(* IEC 61131-3 sources: Industry-PLC-LLM/data/PLCBEAD_repo/PLCBEAD_PLCEmbed-main/PLC-BEAD/Source/OpenPLCv2 (part 5) *)

(* ---- FT_DERIV.ST ---- *)
FUNCTION_BLOCK T_PLC_US_Block
	VAR_OUTPUT
		T_PLC_US :	UDINT;
	END_VAR

	VAR_EXTERNAL
		PLC_TICKS_PER_SEC :	INT;
		PLC_SYS_TICK_CNT :	DINT;
	END_VAR

	VAR
		debug :	BOOL;
		N :	INT;
		Offset :	UDINT;
		temp :	DWORD := DWORD#1;
		mode :	BOOL;
		faktor :	UDINT;
		init :	BOOL;
		v_plc_ticks_per_sec :	UDINT;
		base :	UDINT := UDINT#1000000;
	END_VAR

	IF init = FALSE THEN
		v_plc_ticks_per_sec := INT_TO_UDINT(PLC_TICKS_PER_SEC);
		IF v_plc_ticks_per_sec = UDINT#1024 THEN
			faktor := UDINT#1000;
			mode := FALSE;
		ELSIF v_plc_ticks_per_sec > UDINT#0 THEN
			IF v_plc_ticks_per_sec <= base THEN
				faktor := base / v_plc_ticks_per_sec;
				mode := FALSE;
			ELSE
				faktor := v_plc_ticks_per_sec / base;
				mode := TRUE;
			END_IF;
		ELSE
			faktor := UDINT#1;
		END_IF;
		init := TRUE;
	END_IF;

	IF mode THEN
		T_PLC_US := DINT_TO_UDINT(PLC_SYS_TICK_CNT) / faktor;
	ELSE
		T_PLC_US := DINT_TO_UDINT(PLC_SYS_TICK_CNT) * faktor;
	END_IF;

	IF debug THEN
		T_PLC_US := (DWORD_TO_UDINT(SHL(UDINT_TO_DWORD(T_PLC_US),N) OR SHL(temp,N)) - UDINT#1) + Offset;
	END_IF;
END_FUNCTION_BLOCK

FUNCTION_BLOCK FT_DERIV
	VAR_INPUT
		IN :	REAL;
		K :	REAL := 1.0;
		RUN :	BOOL := TRUE;
	END_VAR

	VAR_OUTPUT
		OUT :	REAL;
	END_VAR

	VAR
		old :	REAL;
		tx :	UDINT;
		last :	UDINT;
		init :	BOOL;
		tc :	REAL;
		T_PLC_US :	T_PLC_US_Block;
	END_VAR

	T_PLC_US();
	tx:= T_PLC_US.T_PLC_US;
	tc := UDINT_TO_REAL(tx - last);

	IF NOT init THEN
		init := TRUE;
		old := in;
	ELSIF run AND tc > 0.0 THEN
		out := (in - old) / tc * 1000000.0 * K;
		old := in;
	ELSE
		out := 0.0;
	END_IF;

	last := tx;

	T_PLC_US();
	tx:= T_PLC_US.T_PLC_US;

	IF NOT init THEN
		init := TRUE;
	ELSIF run AND tx - last > UDINT#0 THEN
		out := (in - old) / UDINT_TO_REAL(tx - last) * 1000000.0 * K;
	ELSE
		out := 0.0;
	END_IF;
	old := in;
	last := tx;
END_FUNCTION_BLOCK

PROGRAM program0
  VAR
	IN  :	REAL;
	K   :	REAL;
	RUN :	BOOL;

	OUT :	REAL;

	func_block : FT_DERIV;
  END_VAR
	func_block.IN :=IN ;
	func_block.K  :=K  ;
	func_block.RUN:=RUN;
	func_block();
	OUT := func_block.OUT;
END_PROGRAM

CONFIGURATION Config0
	VAR_GLOBAL
		PLC_TICKS_PER_SEC :	INT;
		PLC_SYS_TICK_CNT :	DINT;
	END_VAR

	RESOURCE Res0 ON PLC
		TASK task0(INTERVAL := T#20ms,PRIORITY := 0);
		PROGRAM instance0 WITH task0 : program0;
	END_RESOURCE
END_CONFIGURATION

(* ---- FT_IMP.ST ---- *)
FUNCTION_BLOCK T_PLC_US_Block

	VAR_OUTPUT
		T_PLC_US :	UDINT;
	END_VAR

	VAR_EXTERNAL
		PLC_TICKS_PER_SEC :	INT;
		PLC_SYS_TICK_CNT :	DINT;
	END_VAR

	VAR
		debug :	BOOL;
		N :	INT;
		Offset :	UDINT;
		temp :	DWORD := DWORD#1;
		mode :	BOOL;
		faktor :	UDINT;
		init :	BOOL;
		v_plc_ticks_per_sec :	UDINT;
		base :	UDINT := UDINT#1000000;
	END_VAR

	IF init = FALSE THEN
		v_plc_ticks_per_sec := INT_TO_UDINT(PLC_TICKS_PER_SEC);
		IF v_plc_ticks_per_sec = UDINT#1024 THEN
			faktor := UDINT#1000;
			mode := FALSE;
		ELSIF v_plc_ticks_per_sec > UDINT#0 THEN
			IF v_plc_ticks_per_sec <= base THEN
				faktor := base / v_plc_ticks_per_sec;
				mode := FALSE;
			ELSE
				faktor := v_plc_ticks_per_sec / base;
				mode := TRUE;
			END_IF;
		ELSE
			faktor := UDINT#1;
		END_IF;
		init := TRUE;
	END_IF;

	IF mode THEN
		T_PLC_US := DINT_TO_UDINT(PLC_SYS_TICK_CNT) / faktor;
	ELSE
		T_PLC_US := DINT_TO_UDINT(PLC_SYS_TICK_CNT) * faktor;
	END_IF;

	IF debug THEN
		T_PLC_US := (DWORD_TO_UDINT(SHL(UDINT_TO_DWORD(T_PLC_US),N) OR SHL(temp,N)) - UDINT#1) + Offset;
	END_IF;

END_FUNCTION_BLOCK

FUNCTION_BLOCK FT_PT1

	VAR_INPUT
		IN :	REAL;
		T :	TIME;
		K :	REAL := 1.0;
	END_VAR

	VAR_OUTPUT
		OUT :	REAL;
	END_VAR

	VAR
		last :	UDINT;
		tx :	UDINT;
		init :	BOOL;
		T_PLC_US :	T_PLC_US_Block;
	END_VAR

	T_PLC_US();
	tx:= T_PLC_US.T_PLC_US;

	IF NOT init OR T = t#0s THEN
		init := TRUE;
		out := K * in;
	ELSE
		out := out + (in * K - out) * UDINT_TO_REAL(Tx - last) / TIME_TO_REAL(T) * 1.0E-3;
		IF ABS(out) < 1.0E-20 THEN out := 0.0; END_IF;
	END_IF;
	last := tx;

END_FUNCTION_BLOCK

FUNCTION_BLOCK FT_IMP

	VAR_INPUT
		IN :	REAL;
		T :	TIME;
		K :	REAL := 1.0;
	END_VAR

	VAR_OUTPUT
		OUT :	REAL;
	END_VAR

	VAR
		t1 :	FT_PT1;
	END_VAR

	T1(in:= in, T:=T);
	out := (in - t1.out) * K;

END_FUNCTION_BLOCK

PROGRAM program0
  VAR
	IN :	REAL;
	T :	TIME;
	K :	REAL;

	OUT :	REAL;

	func_block : FT_IMP;
  END_VAR
	func_block.IN :=IN ;
	func_block.T  :=T  ;
	func_block.K  :=K  ;
	func_block();
	OUT := func_block.OUT;
END_PROGRAM

CONFIGURATION Config0

	VAR_GLOBAL
		PLC_TICKS_PER_SEC :	INT;
		PLC_SYS_TICK_CNT :	DINT;
	END_VAR

	RESOURCE Res0 ON PLC
		TASK task0(INTERVAL := T#20ms,PRIORITY := 0);
		PROGRAM instance0 WITH task0 : program0;
	END_RESOURCE

END_CONFIGURATION

(* ---- FT_INT.ST ---- *)
FUNCTION_BLOCK T_PLC_MS_block
	VAR_OUTPUT
		T_PLC_MS :	UDINT;
	END_VAR

	VAR_EXTERNAL
		PLC_TICKS_PER_SEC :	INT;
		PLC_SYS_TICK_CNT :	DINT;
	END_VAR

	VAR
		debug :	BOOL;(*Debug-Mode ON / OFF*)
		N :	INT;(*Debug-Faktor*)
		Offset :	UDINT;(*Debug-Offset*)
		temp :	DWORD := DWORD#1;(*Debug-Offset*)
		mode :	BOOL;(*modus*)
		faktor :	UDINT;(*Systemtakt-Faktor*)
		init :	BOOL;
		v_plc_ticks_per_sec :	UDINT;
		base :	UDINT := UDINT#1000;
	END_VAR

	IF init = FALSE THEN
		v_plc_ticks_per_sec := INT_TO_UDINT(PLC_TICKS_PER_SEC);
		IF v_plc_ticks_per_sec = UDINT#1024 THEN
			faktor := UDINT#1;
			mode := FALSE;
		ELSIF v_plc_ticks_per_sec > UDINT#0 THEN
			IF v_plc_ticks_per_sec <= base THEN
				faktor := base / v_plc_ticks_per_sec;
				mode := FALSE;
			ELSE
				faktor := v_plc_ticks_per_sec / base;
				mode := TRUE;
			END_IF;
		ELSE
			faktor := UDINT#1;
		END_IF;
		init := TRUE;
	END_IF;

	IF mode THEN
		T_PLC_MS := DINT_TO_UDINT(PLC_SYS_TICK_CNT) / faktor;
	ELSE
		T_PLC_MS := DINT_TO_UDINT(PLC_SYS_TICK_CNT) * faktor;
	END_IF;

	IF debug THEN
		T_PLC_MS := (DWORD_TO_UDINT(SHL(UDINT_TO_DWORD(T_PLC_MS),N) OR SHL(temp,N)) - UDINT#1) + Offset;
	END_IF;
END_FUNCTION_BLOCK

FUNCTION_BLOCK INTEGRATE

	VAR_INPUT
		E :	BOOL := TRUE;
		X :	REAL;
		K :	REAL := 1.0;
	END_VAR

	VAR_IN_OUT
		Y :	REAL;
	END_VAR

	VAR
		X_last :	REAL;
		init :	BOOL;
		T_PLC_MS :	T_PLC_MS_block;
		last :	UDINT;
		tx :	UDINT;
	END_VAR

	T_PLC_MS();
	tx:= T_PLC_MS.T_PLC_MS;

	IF NOT init THEN
		init := TRUE;
		X_last := X;
	ELSIF E THEN
		Y := (X + X_LAST) * 0.5E-3 * UDINT_TO_REAL(tx-last) * K + Y;
		X_last := X;
	END_IF;
	last := tx;

END_FUNCTION_BLOCK

FUNCTION_BLOCK FT_INT_Block

	VAR_INPUT
		IN :	REAL;
		K :	REAL := 1.0;
		RUN :	BOOL := TRUE;
		RST :	BOOL;
		OUT_MIN :	REAL := REAL#-1.0E-37;
		OUT_MAX :	REAL := REAL#1.0E37;
	END_VAR

	VAR_OUTPUT
		OUT :	REAL;
		LIM :	BOOL;
	END_VAR

	VAR
		INTEG :	INTEGRATE;
	END_VAR

	IF rst THEN
		out := 0.0;
	ELSE
		integ(X := IN, E := RUN, K := K, Y := out);
		out := integ.Y;
	END_IF;

	(* limit the outputs *)
	IF out >= OUT_MAX THEN
		out := out_max;
		LIM := TRUE;
	ELSIF out <= out_min THEN
		out := out_min;
		lim := TRUE;
	ELSE
		lim := FALSE;
	END_IF;

END_FUNCTION_BLOCK

PROGRAM program0
  VAR
	IN :	REAL;
	K :	REAL := 1.0;
	RUN :	BOOL := TRUE;
	RST :	BOOL;
	OUT_MIN :	REAL := REAL#-1.0E-37;
	OUT_MAX :	REAL := REAL#1.0E37;

	OUT :	REAL;
	LIM :	BOOL;

	func_block : FT_INT_Block;
  END_VAR
	func_block.IN :=IN ;
	func_block.K :=K  ;
	func_block.RUN :=RUN  ;
	func_block.RST :=RST ;
	func_block.OUT_MIN :=OUT_MIN  ;
	func_block.OUT_MAX :=OUT_MAX  ;
	func_block();
	OUT := func_block.OUT;
	LIM := func_block.LIM;
END_PROGRAM

CONFIGURATION Config0

	VAR_GLOBAL
		PLC_TICKS_PER_SEC :	INT;
		PLC_SYS_TICK_CNT :	DINT;
	END_VAR

	RESOURCE Res0 ON PLC
		TASK task0(INTERVAL := T#20ms,PRIORITY := 0);
		PROGRAM instance0 WITH task0 : program0;
	END_RESOURCE

END_CONFIGURATION

(* ---- FT_MIN_MAX.ST ---- *)
FUNCTION_BLOCK FT_MIN_MAX_Block

  VAR_INPUT
    IN :	REAL;
    RST :	BOOL;
  END_VAR

  VAR_OUTPUT
    MX :	REAL;
    MN :	REAL;
  END_VAR

  VAR
    init :	BOOL;
  END_VAR

  IF (rst = TRUE) OR (init = FALSE) THEN
    mn := in;
    mx := in;
    init := TRUE;
  ELSIF (in < mn) THEN
    mn := in;
  ELSIF (in > mx) THEN
    mx := in;
  END_IF;

END_FUNCTION_BLOCK

PROGRAM program0
  VAR
    IN :	REAL;
    RST :	BOOL;

	  MX :	REAL;
    MN :	REAL;

  	func_block : FT_MIN_MAX_Block;
  END_VAR

	func_block.IN :=IN;
	func_block.RST := RST;
	func_block();
	MX := func_block.MX;
	MN := func_block.MN;

END_PROGRAM

CONFIGURATION Config0

	VAR_GLOBAL
		PLC_TICKS_PER_SEC :	INT;
		PLC_SYS_TICK_CNT :	DINT;
	END_VAR

	RESOURCE Res0 ON PLC
		TASK task0(INTERVAL := T#20ms,PRIORITY := 0);
		PROGRAM instance0 WITH task0 : program0;
	END_RESOURCE

END_CONFIGURATION

(* ---- FT_PD.ST ---- *)
FUNCTION_BLOCK T_PLC_US_Block
	VAR_OUTPUT
		T_PLC_US :	UDINT;
	END_VAR

	VAR_EXTERNAL
		PLC_TICKS_PER_SEC :	INT;
		PLC_SYS_TICK_CNT :	DINT;
	END_VAR

	VAR
		debug :	BOOL;
		N :	INT;
		Offset :	UDINT;
		temp :	DWORD := DWORD#1;
		mode :	BOOL;
		faktor :	UDINT;
		init :	BOOL;
		v_plc_ticks_per_sec :	UDINT;
		base :	UDINT := UDINT#1000000;
	END_VAR

	IF init = FALSE THEN
		v_plc_ticks_per_sec := INT_TO_UDINT(PLC_TICKS_PER_SEC);
		IF v_plc_ticks_per_sec = UDINT#1024 THEN
			faktor := UDINT#1000;
			mode := FALSE;
		ELSIF v_plc_ticks_per_sec > UDINT#0 THEN
			IF v_plc_ticks_per_sec <= base THEN
				faktor := base / v_plc_ticks_per_sec;
				mode := FALSE;
			ELSE
				faktor := v_plc_ticks_per_sec / base;
				mode := TRUE;
			END_IF;
		ELSE
			faktor := UDINT#1;
		END_IF;
		init := TRUE;
	END_IF;

	IF mode THEN
		T_PLC_US := DINT_TO_UDINT(PLC_SYS_TICK_CNT) / faktor;
	ELSE
		T_PLC_US := DINT_TO_UDINT(PLC_SYS_TICK_CNT) * faktor;
	END_IF;

	IF debug THEN
		T_PLC_US := (DWORD_TO_UDINT(SHL(UDINT_TO_DWORD(T_PLC_US),N) OR SHL(temp,N)) - UDINT#1) + Offset;
	END_IF;
END_FUNCTION_BLOCK

FUNCTION_BLOCK FT_DERIV
	VAR_INPUT
		IN :	REAL;
		K :	REAL := 1.0;
		RUN :	BOOL := TRUE;
	END_VAR

	VAR_OUTPUT
		OUT :	REAL;
	END_VAR

	VAR
		old :	REAL;
		tx :	UDINT;
		last :	UDINT;
		init :	BOOL;
		tc :	REAL;
		T_PLC_US :	T_PLC_US_Block;
	END_VAR

	T_PLC_US();
	tx:= T_PLC_US.T_PLC_US;
	tc := UDINT_TO_REAL(tx - last);

	IF NOT init THEN
		init := TRUE;
		old := in;
	ELSIF run AND tc > 0.0 THEN
		out := (in - old) / tc * 1000000.0 * K;
		old := in;
	ELSE
		out := 0.0;
	END_IF;

	last := tx;

	T_PLC_US();
	tx:= T_PLC_US.T_PLC_US;

	IF NOT init THEN
		init := TRUE;
	ELSIF run AND tx - last > UDINT#0 THEN
		out := (in - old) / UDINT_TO_REAL(tx - last) * 1000000.0 * K;
	ELSE
		out := 0.0;
	END_IF;
	old := in;
	last := tx;
END_FUNCTION_BLOCK

FUNCTION_BLOCK FT_PD_Block

	VAR_INPUT
		IN :	REAL;
		KP :	REAL := 1.0;
		TV :	REAL := 1.0;
	END_VAR

	VAR_OUTPUT
		Y :	REAL;
	END_VAR

	VAR
		diff :	FT_DERIV;
	END_VAR

	diff(IN := IN, K := TV);

	Y := KP * (diff.out + IN);

END_FUNCTION_BLOCK

PROGRAM program0
	VAR
		IN :	REAL;
		KP :	REAL := 1.0;
		TV :	REAL := 1.0;
		Y :	REAL;
		func_block : FT_PD_Block;
	END_VAR
	func_block.IN :=IN;
	func_block.KP :=KP;
	func_block.TV :=TV;
	func_block();
	Y := func_block.Y;
END_PROGRAM

CONFIGURATION Config0

	VAR_GLOBAL
		PLC_TICKS_PER_SEC :	INT;
		PLC_SYS_TICK_CNT :	DINT;
	END_VAR

	RESOURCE Res0 ON PLC
		TASK task0(INTERVAL := T#20ms,PRIORITY := 0);
		PROGRAM instance0 WITH task0 : program0;
	END_RESOURCE

END_CONFIGURATION

(* ---- FT_PDT1.ST ---- *)
FUNCTION _REAL_TO_UDINT:UDINT
  VAR_INPUT
    X :	REAL;
  END_VAR

  IF REAL_TO_UDINT(0.5) = UDINT#1 THEN
    _REAL_TO_UDINT := REAL_TO_UDINT(x);
  ELSIF X > 0.0 THEN
    _REAL_TO_UDINT := REAL_TO_UDINT(x+0.5);
  ELSIF X < 0.0 THEN
    _REAL_TO_UDINT := REAL_TO_UDINT(x-0.5);
  ELSE
    _REAL_TO_UDINT := UDINT#0;
  END_IF;
END_FUNCTION

FUNCTION REAL_TO_TIME2:TIME
	VAR_INPUT
		IN :	REAL;
	END_VAR

	REAL_TO_TIME2 := DINT_TO_TIME(UDINT_TO_DINT(_REAL_TO_UDINT(IN)));
END_FUNCTION

FUNCTION_BLOCK T_PLC_US_Block
	VAR_OUTPUT
		T_PLC_US :	UDINT;
	END_VAR

	VAR_EXTERNAL
		PLC_TICKS_PER_SEC :	INT;
		PLC_SYS_TICK_CNT :	DINT;
	END_VAR

	VAR
		debug :	BOOL;
		N :	INT;
		Offset :	UDINT;
		temp :	DWORD := DWORD#1;
		mode :	BOOL;
		faktor :	UDINT;
		init :	BOOL;
		v_plc_ticks_per_sec :	UDINT;
		base :	UDINT := UDINT#1000000;
	END_VAR

	IF init = FALSE THEN
		v_plc_ticks_per_sec := INT_TO_UDINT(PLC_TICKS_PER_SEC);
		IF v_plc_ticks_per_sec = UDINT#1024 THEN
			faktor := UDINT#1000;
			mode := FALSE;
		ELSIF v_plc_ticks_per_sec > UDINT#0 THEN
			IF v_plc_ticks_per_sec <= base THEN
				faktor := base / v_plc_ticks_per_sec;
				mode := FALSE;
			ELSE
				faktor := v_plc_ticks_per_sec / base;
				mode := TRUE;
			END_IF;
		ELSE
			faktor := UDINT#1;
		END_IF;
		init := TRUE;
	END_IF;

	IF mode THEN
		T_PLC_US := DINT_TO_UDINT(PLC_SYS_TICK_CNT) / faktor;
	ELSE
		T_PLC_US := DINT_TO_UDINT(PLC_SYS_TICK_CNT) * faktor;
	END_IF;

	IF debug THEN
		T_PLC_US := (DWORD_TO_UDINT(SHL(UDINT_TO_DWORD(T_PLC_US),N) OR SHL(temp,N)) - UDINT#1) + Offset;
	END_IF;
END_FUNCTION_BLOCK

FUNCTION_BLOCK FT_DERIV
	VAR_INPUT
		IN :	REAL;
		K :	REAL := 1.0;
		RUN :	BOOL := TRUE;
	END_VAR

	VAR_OUTPUT
		OUT :	REAL;
	END_VAR

	VAR
		old :	REAL;
		tx :	UDINT;
		last :	UDINT;
		init :	BOOL;
		tc :	REAL;
		T_PLC_US :	T_PLC_US_Block;
	END_VAR

	T_PLC_US();
	tx:= T_PLC_US.T_PLC_US;
	tc := UDINT_TO_REAL(tx - last);

	IF NOT init THEN
		init := TRUE;
		old := in;
	ELSIF run AND tc > 0.0 THEN
		out := (in - old) / tc * 1000000.0 * K;
		old := in;
	ELSE
		out := 0.0;
	END_IF;

	last := tx;

	T_PLC_US();
	tx:= T_PLC_US.T_PLC_US;

	IF NOT init THEN
		init := TRUE;
	ELSIF run AND tx - last > UDINT#0 THEN
		out := (in - old) / UDINT_TO_REAL(tx - last) * 1000000.0 * K;
	ELSE
		out := 0.0;
	END_IF;
	old := in;
	last := tx;
END_FUNCTION_BLOCK

FUNCTION_BLOCK FT_PT1

	VAR_INPUT
		IN :	REAL;
		T :	TIME;
		K :	REAL := 1.0;
	END_VAR

	VAR_OUTPUT
		OUT :	REAL;
	END_VAR

	VAR
		last :	UDINT;
		tx :	UDINT;
		init :	BOOL;
		T_PLC_US :	T_PLC_US_Block;
	END_VAR

	T_PLC_US();
	tx:= T_PLC_US.T_PLC_US;

	IF NOT init OR T = t#0s THEN
		init := TRUE;
		out := K * in;
	ELSE
		out := out + (in * K - out) * UDINT_TO_REAL(Tx - last) / TIME_TO_REAL(T) * 1.0E-3;
		IF ABS(out) < 1.0E-20 THEN out := 0.0; END_IF;
	END_IF;
	last := tx;
END_FUNCTION_BLOCK

FUNCTION_BLOCK FT_PDT1_Block

	VAR_INPUT
		IN :	REAL;
		KP :	REAL := 1.0;
		TV :	REAL := 1.0;
		T1 :	REAL := 1.0;
	END_VAR

	VAR_OUTPUT
		Y :	REAL;
	END_VAR

	VAR
		diff :	FT_DERIV;
		_TP :	FT_PT1;
	END_VAR

	diff(IN := IN, K := TV);

	_tp(in := diff.out, T := REAL_TO_TIME2(T1));

	Y := KP * (_tp.out + IN);

END_FUNCTION_BLOCK

PROGRAM program0
	VAR
		IN :	REAL;
		KP :	REAL := 1.0;
		TV :	REAL := 1.0;
		T1 :	REAL := 1.0;

		Y :	REAL;
		func_block : FT_PDT1_Block;
	END_VAR
	func_block.IN :=IN;
	func_block.KP :=KP;
	func_block.TV :=TV;
	func_block.T1 :=T1;
	func_block();
	Y := func_block.Y;
END_PROGRAM

CONFIGURATION Config0

	VAR_GLOBAL
		PLC_TICKS_PER_SEC :	INT;
		PLC_SYS_TICK_CNT :	DINT;
	END_VAR

	RESOURCE Res0 ON PLC
		TASK task0(INTERVAL := T#20ms,PRIORITY := 0);
		PROGRAM instance0 WITH task0 : program0;
	END_RESOURCE

END_CONFIGURATION

(* ---- FT_PI.ST ---- *)
FUNCTION_BLOCK T_PLC_MS_block
	VAR_OUTPUT
		T_PLC_MS :	UDINT;
	END_VAR

	VAR_EXTERNAL
		PLC_TICKS_PER_SEC :	INT;
		PLC_SYS_TICK_CNT :	DINT;
	END_VAR

	VAR
		debug :	BOOL;(*Debug-Mode ON / OFF*)
		N :	INT;(*Debug-Faktor*)
		Offset :	UDINT;(*Debug-Offset*)
		temp :	DWORD := DWORD#1;(*Debug-Offset*)
		mode :	BOOL;(*modus*)
		faktor :	UDINT;(*Systemtakt-Faktor*)
		init :	BOOL;
		v_plc_ticks_per_sec :	UDINT;
		base :	UDINT := UDINT#1000;
	END_VAR

	IF init = FALSE THEN
		v_plc_ticks_per_sec := INT_TO_UDINT(PLC_TICKS_PER_SEC);
		IF v_plc_ticks_per_sec = UDINT#1024 THEN
			faktor := UDINT#1;
			mode := FALSE;
		ELSIF v_plc_ticks_per_sec > UDINT#0 THEN
			IF v_plc_ticks_per_sec <= base THEN
				faktor := base / v_plc_ticks_per_sec;
				mode := FALSE;
			ELSE
				faktor := v_plc_ticks_per_sec / base;
				mode := TRUE;
			END_IF;
		ELSE
			faktor := UDINT#1;
		END_IF;
		init := TRUE;
	END_IF;

	IF mode THEN
		T_PLC_MS := DINT_TO_UDINT(PLC_SYS_TICK_CNT) / faktor;
	ELSE
		T_PLC_MS := DINT_TO_UDINT(PLC_SYS_TICK_CNT) * faktor;
	END_IF;

	IF debug THEN
		T_PLC_MS := (DWORD_TO_UDINT(SHL(UDINT_TO_DWORD(T_PLC_MS),N) OR SHL(temp,N)) - UDINT#1) + Offset;
	END_IF;
END_FUNCTION_BLOCK

FUNCTION_BLOCK INTEGRATE

	VAR_INPUT
		E :	BOOL := TRUE;
		X :	REAL;
		K :	REAL := 1.0;
	END_VAR

	VAR_IN_OUT
		Y :	REAL;
	END_VAR

	VAR
		X_last :	REAL;
		init :	BOOL;
		T_PLC_MS :	T_PLC_MS_block;
		last :	UDINT;
		tx :	UDINT;
	END_VAR

	T_PLC_MS();
	tx:= T_PLC_MS.T_PLC_MS;

	IF NOT init THEN
		init := TRUE;
		X_last := X;
	ELSIF E THEN
		Y := (X + X_LAST) * 0.5E-3 * UDINT_TO_REAL(tx-last) * K + Y;
		X_last := X;
	END_IF;
	last := tx;

END_FUNCTION_BLOCK

FUNCTION_BLOCK FT_INT_Block

	VAR_INPUT
		IN :	REAL;
		K :	REAL := 1.0;
		RUN :	BOOL := TRUE;
		RST :	BOOL;
		OUT_MIN :	REAL := REAL#-1.0E-37;
		OUT_MAX :	REAL := REAL#1.0E37;
	END_VAR

	VAR_OUTPUT
		OUT :	REAL;
		LIM :	BOOL;
	END_VAR

	VAR
		INTEG :	INTEGRATE;
	END_VAR

	IF rst THEN
		out := 0.0;
	ELSE
		integ(X := IN, E := RUN, K := K, Y := out);
		out := integ.Y;
	END_IF;

	(* limit the outputs *)
	IF out >= OUT_MAX THEN
		out := out_max;
		LIM := TRUE;
	ELSIF out <= out_min THEN
		out := out_min;
		lim := TRUE;
	ELSE
		lim := FALSE;
	END_IF;

END_FUNCTION_BLOCK

FUNCTION_BLOCK FT_PI

	VAR_INPUT
		IN :	REAL;
		KP :	REAL := 1.0;
		KI :	REAL := 1.0;
		ILIM_L :	REAL := -1.0E38;
		ILIM_H :	REAL := 1.0E38;
		IEN :	BOOL := TRUE;
		RST :	BOOL := FALSE;
	END_VAR

	VAR_OUTPUT
		Y :	REAL;
		LIM :	BOOL;
	END_VAR

	VAR
		integ :	FT_INT_Block;
	END_VAR

	integ(IN := IN, K := KI, RUN := IEN, RST := RST, OUT_MIN := ILIM_L, OUT_MAX := ILIM_H);
	(* check if integrator has reached its limits and set overflow *)
	LIM := integ.LIM;
	Y := KP * IN + integ.Out;

END_FUNCTION_BLOCK

PROGRAM program0
	VAR
		IN :	REAL;
		KP :	REAL := 1.0;
		KI :	REAL := 1.0;
		ILIM_L :	REAL := -1.0E38;
		ILIM_H :	REAL := 1.0E38;
		IEN :	BOOL := TRUE;
		RST :	BOOL := FALSE;

		Y :	REAL;
		LIM :	BOOL;

		func_block : FT_PI;
	END_VAR
	func_block.IN :=IN;
	func_block.KP :=KP;
	func_block.KI :=KI;
	func_block.ILIM_L :=ILIM_L;
	func_block.ILIM_H :=ILIM_H;
	func_block.IEN :=IEN;
	func_block.RST :=RST;

	func_block();
	Y := func_block.Y;
	LIM := func_block.LIM;
END_PROGRAM

CONFIGURATION Config0

	VAR_GLOBAL
		PLC_TICKS_PER_SEC :	INT;
		PLC_SYS_TICK_CNT :	DINT;
	END_VAR

	RESOURCE Res0 ON PLC
		TASK task0(INTERVAL := T#20ms,PRIORITY := 0);
		PROGRAM instance0 WITH task0 : program0;
	END_RESOURCE

END_CONFIGURATION

(* ---- FT_PID.ST ---- *)
FUNCTION_BLOCK T_PLC_US_Block
	VAR_OUTPUT
		T_PLC_US :	UDINT;
	END_VAR

	VAR_EXTERNAL
		PLC_TICKS_PER_SEC :	INT;
		PLC_SYS_TICK_CNT :	DINT;
	END_VAR

	VAR
		debug :	BOOL;
		N :	INT;
		Offset :	UDINT;
		temp :	DWORD := DWORD#1;
		mode :	BOOL;
		faktor :	UDINT;
		init :	BOOL;
		v_plc_ticks_per_sec :	UDINT;
		base :	UDINT := UDINT#1000000;
	END_VAR

	IF init = FALSE THEN
		v_plc_ticks_per_sec := INT_TO_UDINT(PLC_TICKS_PER_SEC);
		IF v_plc_ticks_per_sec = UDINT#1024 THEN
			faktor := UDINT#1000;
			mode := FALSE;
		ELSIF v_plc_ticks_per_sec > UDINT#0 THEN
			IF v_plc_ticks_per_sec <= base THEN
				faktor := base / v_plc_ticks_per_sec;
				mode := FALSE;
			ELSE
				faktor := v_plc_ticks_per_sec / base;
				mode := TRUE;
			END_IF;
		ELSE
			faktor := UDINT#1;
		END_IF;
		init := TRUE;
	END_IF;

	IF mode THEN
		T_PLC_US := DINT_TO_UDINT(PLC_SYS_TICK_CNT) / faktor;
	ELSE
		T_PLC_US := DINT_TO_UDINT(PLC_SYS_TICK_CNT) * faktor;
	END_IF;

	IF debug THEN
		T_PLC_US := (DWORD_TO_UDINT(SHL(UDINT_TO_DWORD(T_PLC_US),N) OR SHL(temp,N)) - UDINT#1) + Offset;
	END_IF;
END_FUNCTION_BLOCK

FUNCTION_BLOCK T_PLC_MS_block
	VAR_OUTPUT
		T_PLC_MS :	UDINT;
	END_VAR

	VAR_EXTERNAL
		PLC_TICKS_PER_SEC :	INT;
		PLC_SYS_TICK_CNT :	DINT;
	END_VAR

	VAR
		debug :	BOOL;(*Debug-Mode ON / OFF*)
		N :	INT;(*Debug-Faktor*)
		Offset :	UDINT;(*Debug-Offset*)
		temp :	DWORD := DWORD#1;(*Debug-Offset*)
		mode :	BOOL;(*modus*)
		faktor :	UDINT;(*Systemtakt-Faktor*)
		init :	BOOL;
		v_plc_ticks_per_sec :	UDINT;
		base :	UDINT := UDINT#1000;
	END_VAR

	IF init = FALSE THEN
		v_plc_ticks_per_sec := INT_TO_UDINT(PLC_TICKS_PER_SEC);
		IF v_plc_ticks_per_sec = UDINT#1024 THEN
			faktor := UDINT#1;
			mode := FALSE;
		ELSIF v_plc_ticks_per_sec > UDINT#0 THEN
			IF v_plc_ticks_per_sec <= base THEN
				faktor := base / v_plc_ticks_per_sec;
				mode := FALSE;
			ELSE
				faktor := v_plc_ticks_per_sec / base;
				mode := TRUE;
			END_IF;
		ELSE
			faktor := UDINT#1;
		END_IF;
		init := TRUE;
	END_IF;

	IF mode THEN
		T_PLC_MS := DINT_TO_UDINT(PLC_SYS_TICK_CNT) / faktor;
	ELSE
		T_PLC_MS := DINT_TO_UDINT(PLC_SYS_TICK_CNT) * faktor;
	END_IF;

	IF debug THEN
		T_PLC_MS := (DWORD_TO_UDINT(SHL(UDINT_TO_DWORD(T_PLC_MS),N) OR SHL(temp,N)) - UDINT#1) + Offset;
	END_IF;
END_FUNCTION_BLOCK

FUNCTION_BLOCK INTEGRATE

	VAR_INPUT
		E :	BOOL := TRUE;
		X :	REAL;
		K :	REAL := 1.0;
	END_VAR

	VAR_IN_OUT
		Y :	REAL;
	END_VAR

	VAR
		X_last :	REAL;
		init :	BOOL;
		T_PLC_MS :	T_PLC_MS_block;
		last :	UDINT;
		tx :	UDINT;
	END_VAR

	T_PLC_MS();
	tx:= T_PLC_MS.T_PLC_MS;

	IF NOT init THEN
		init := TRUE;
		X_last := X;
	ELSIF E THEN
		Y := (X + X_LAST) * 0.5E-3 * UDINT_TO_REAL(tx-last) * K + Y;
		X_last := X;
	END_IF;
	last := tx;

END_FUNCTION_BLOCK

FUNCTION_BLOCK FT_INT_Block

	VAR_INPUT
		IN :	REAL;
		K :	REAL := 1.0;
		RUN :	BOOL := TRUE;
		RST :	BOOL;
		OUT_MIN :	REAL := REAL#-1.0E-37;
		OUT_MAX :	REAL := REAL#1.0E37;
	END_VAR

	VAR_OUTPUT
		OUT :	REAL;
		LIM :	BOOL;
	END_VAR

	VAR
		INTEG :	INTEGRATE;
	END_VAR

	IF rst THEN
		out := 0.0;
	ELSE
		integ(X := IN, E := RUN, K := K, Y := out);
		out := integ.Y;
	END_IF;

	(* limit the outputs *)
	IF out >= OUT_MAX THEN
		out := out_max;
		LIM := TRUE;
	ELSIF out <= out_min THEN
		out := out_min;
		lim := TRUE;
	ELSE
		lim := FALSE;
	END_IF;

END_FUNCTION_BLOCK

FUNCTION_BLOCK FT_DERIV
	VAR_INPUT
		IN :	REAL;
		K :	REAL := 1.0;
		RUN :	BOOL := TRUE;
	END_VAR

	VAR_OUTPUT
		OUT :	REAL;
	END_VAR

	VAR
		old :	REAL;
		tx :	UDINT;
		last :	UDINT;
		init :	BOOL;
		tc :	REAL;
		T_PLC_US :	T_PLC_US_Block;
	END_VAR

	T_PLC_US();
	tx:= T_PLC_US.T_PLC_US;
	tc := UDINT_TO_REAL(tx - last);

	IF NOT init THEN
		init := TRUE;
		old := in;
	ELSIF run AND tc > 0.0 THEN
		out := (in - old) / tc * 1000000.0 * K;
		old := in;
	ELSE
		out := 0.0;
	END_IF;

	last := tx;

	T_PLC_US();
	tx:= T_PLC_US.T_PLC_US;

	IF NOT init THEN
		init := TRUE;
	ELSIF run AND tx - last > UDINT#0 THEN
		out := (in - old) / UDINT_TO_REAL(tx - last) * 1000000.0 * K;
	ELSE
		out := 0.0;
	END_IF;
	old := in;
	last := tx;
END_FUNCTION_BLOCK

FUNCTION_BLOCK FT_PID

	VAR_INPUT
		IN :	REAL;
		KP :	REAL := 1.0;
		TN :	REAL := 1.0;
		TV :	REAL := 1.0;
		ILIM_L :	REAL := -1.0E38;
		ILIM_H :	REAL := 1.0E38;
		IEN :	BOOL := TRUE;
		RST :	BOOL := FALSE;
	END_VAR

	VAR_OUTPUT
		Y :	REAL;
		LIM :	BOOL;
	END_VAR

	VAR
		integ :	FT_INT_Block;
		diff :	FT_DERIV;
	END_VAR

	IF TN > 0.0 THEN
		integ(IN := IN, K := 1.0 / TN, RUN := IEN, RST := RST, OUT_MIN := ILIM_L, OUT_MAX := ILIM_H);
	ELSE
		integ(RST := FALSE);
	END_IF;

	(* run differentiator *)
	diff(IN := IN, K := TV);

	(* combine both values *)
	Y := KP * (integ.Out + diff.out + IN);

	(* check if integrator has reached its limits and set overflow *)
	LIM := integ.LIM;

END_FUNCTION_BLOCK

PROGRAM program0
	VAR
		IN :	REAL;
		KP :	REAL := 1.0;
		TN :	REAL := 1.0;
		TV :	REAL := 1.0;
		ILIM_L :	REAL := -1.0E38;
		ILIM_H :	REAL := 1.0E38;
		IEN :	BOOL := TRUE;
		RST :	BOOL := FALSE;

		Y :	REAL;
		LIM :	BOOL;

		func_block : FT_PID;
	END_VAR
	func_block.IN :=IN;
	func_block.KP :=KP;
	func_block.TN :=TN;
	func_block.TV :=TV;
	func_block.ILIM_L :=ILIM_L;
	func_block.ILIM_H :=ILIM_H;
	func_block.IEN :=IEN;
	func_block.RST :=RST;

	func_block();
	Y := func_block.Y;
	LIM := func_block.LIM;
END_PROGRAM

CONFIGURATION Config0

	VAR_GLOBAL
		PLC_TICKS_PER_SEC :	INT;
		PLC_SYS_TICK_CNT :	DINT;
	END_VAR

	RESOURCE Res0 ON PLC
		TASK task0(INTERVAL := T#20ms,PRIORITY := 0);
		PROGRAM instance0 WITH task0 : program0;
	END_RESOURCE

END_CONFIGURATION

(* ---- FT_PIDW.ST ---- *)
FUNCTION _REAL_TO_UDINT:UDINT
  VAR_INPUT
    X :	REAL;
  END_VAR

  IF REAL_TO_UDINT(0.5) = UDINT#1 THEN
    _REAL_TO_UDINT := REAL_TO_UDINT(x);
  ELSIF X > 0.0 THEN
    _REAL_TO_UDINT := REAL_TO_UDINT(x+0.5);
  ELSIF X < 0.0 THEN
    _REAL_TO_UDINT := REAL_TO_UDINT(x-0.5);
  ELSE
    _REAL_TO_UDINT := UDINT#0;
  END_IF;
END_FUNCTION

FUNCTION REAL_TO_TIME2:TIME
	VAR_INPUT
		IN :	REAL;
	END_VAR

	REAL_TO_TIME2 := DINT_TO_TIME(UDINT_TO_DINT(_REAL_TO_UDINT(IN)));
END_FUNCTION

FUNCTION_BLOCK T_PLC_US_Block
	VAR_OUTPUT
		T_PLC_US :	UDINT;
	END_VAR

	VAR_EXTERNAL
		PLC_TICKS_PER_SEC :	INT;
		PLC_SYS_TICK_CNT :	DINT;
	END_VAR

	VAR
		debug :	BOOL;
		N :	INT;
		Offset :	UDINT;
		temp :	DWORD := DWORD#1;
		mode :	BOOL;
		faktor :	UDINT;
		init :	BOOL;
		v_plc_ticks_per_sec :	UDINT;
		base :	UDINT := UDINT#1000000;
	END_VAR

	IF init = FALSE THEN
		v_plc_ticks_per_sec := INT_TO_UDINT(PLC_TICKS_PER_SEC);
		IF v_plc_ticks_per_sec = UDINT#1024 THEN
			faktor := UDINT#1000;
			mode := FALSE;
		ELSIF v_plc_ticks_per_sec > UDINT#0 THEN
			IF v_plc_ticks_per_sec <= base THEN
				faktor := base / v_plc_ticks_per_sec;
				mode := FALSE;
			ELSE
				faktor := v_plc_ticks_per_sec / base;
				mode := TRUE;
			END_IF;
		ELSE
			faktor := UDINT#1;
		END_IF;
		init := TRUE;
	END_IF;

	IF mode THEN
		T_PLC_US := DINT_TO_UDINT(PLC_SYS_TICK_CNT) / faktor;
	ELSE
		T_PLC_US := DINT_TO_UDINT(PLC_SYS_TICK_CNT) * faktor;
	END_IF;

	IF debug THEN
		T_PLC_US := (DWORD_TO_UDINT(SHL(UDINT_TO_DWORD(T_PLC_US),N) OR SHL(temp,N)) - UDINT#1) + Offset;
	END_IF;
END_FUNCTION_BLOCK

FUNCTION_BLOCK FT_DERIV
	VAR_INPUT
		IN :	REAL;
		K :	REAL := 1.0;
		RUN :	BOOL := TRUE;
	END_VAR

	VAR_OUTPUT
		OUT :	REAL;
	END_VAR

	VAR
		old :	REAL;
		tx :	UDINT;
		last :	UDINT;
		init :	BOOL;
		tc :	REAL;
		T_PLC_US :	T_PLC_US_Block;
	END_VAR

	T_PLC_US();
	tx:= T_PLC_US.T_PLC_US;
	tc := UDINT_TO_REAL(tx - last);

	IF NOT init THEN
		init := TRUE;
		old := in;
	ELSIF run AND tc > 0.0 THEN
		out := (in - old) / tc * 1000000.0 * K;
		old := in;
	ELSE
		out := 0.0;
	END_IF;

	last := tx;

	T_PLC_US();
	tx:= T_PLC_US.T_PLC_US;

	IF NOT init THEN
		init := TRUE;
	ELSIF run AND tx - last > UDINT#0 THEN
		out := (in - old) / UDINT_TO_REAL(tx - last) * 1000000.0 * K;
	ELSE
		out := 0.0;
	END_IF;
	old := in;
	last := tx;
END_FUNCTION_BLOCK
FUNCTION_BLOCK T_PLC_MS_block
	VAR_OUTPUT
		T_PLC_MS :	UDINT;
	END_VAR

	VAR_EXTERNAL
		PLC_TICKS_PER_SEC :	INT;
		PLC_SYS_TICK_CNT :	DINT;
	END_VAR

	VAR
		debug :	BOOL;(*Debug-Mode ON / OFF*)
		N :	INT;(*Debug-Faktor*)
		Offset :	UDINT;(*Debug-Offset*)
		temp :	DWORD := DWORD#1;(*Debug-Offset*)
		mode :	BOOL;(*modus*)
		faktor :	UDINT;(*Systemtakt-Faktor*)
		init :	BOOL;
		v_plc_ticks_per_sec :	UDINT;
		base :	UDINT := UDINT#1000;
	END_VAR

	IF init = FALSE THEN
		v_plc_ticks_per_sec := INT_TO_UDINT(PLC_TICKS_PER_SEC);
		IF v_plc_ticks_per_sec = UDINT#1024 THEN
			faktor := UDINT#1;
			mode := FALSE;
		ELSIF v_plc_ticks_per_sec > UDINT#0 THEN
			IF v_plc_ticks_per_sec <= base THEN
				faktor := base / v_plc_ticks_per_sec;
				mode := FALSE;
			ELSE
				faktor := v_plc_ticks_per_sec / base;
				mode := TRUE;
			END_IF;
		ELSE
			faktor := UDINT#1;
		END_IF;
		init := TRUE;
	END_IF;

	IF mode THEN
		T_PLC_MS := DINT_TO_UDINT(PLC_SYS_TICK_CNT) / faktor;
	ELSE
		T_PLC_MS := DINT_TO_UDINT(PLC_SYS_TICK_CNT) * faktor;
	END_IF;

	IF debug THEN
		T_PLC_MS := (DWORD_TO_UDINT(SHL(UDINT_TO_DWORD(T_PLC_MS),N) OR SHL(temp,N)) - UDINT#1) + Offset;
	END_IF;
END_FUNCTION_BLOCK

FUNCTION_BLOCK INTEGRATE

	VAR_INPUT
		E :	BOOL := TRUE;
		X :	REAL;
		K :	REAL := 1.0;
	END_VAR

	VAR_IN_OUT
		Y :	REAL;
	END_VAR

	VAR
		X_last :	REAL;
		init :	BOOL;
		T_PLC_MS :	T_PLC_MS_block;
		last :	UDINT;
		tx :	UDINT;
	END_VAR

	T_PLC_MS();
	tx:= T_PLC_MS.T_PLC_MS;

	IF NOT init THEN
		init := TRUE;
		X_last := X;
	ELSIF E THEN
		Y := (X + X_LAST) * 0.5E-3 * UDINT_TO_REAL(tx-last) * K + Y;
		X_last := X;
	END_IF;
	last := tx;

END_FUNCTION_BLOCK

FUNCTION_BLOCK FT_PIDW

	VAR_INPUT
		IN :	REAL;
		KP :	REAL := 1.0;
		TN :	REAL := 1.0;
		TV :	REAL := 1.0;
		LIM_L :	REAL := -1.0E38;
		LIM_H :	REAL := 1.0E38;
		RST :	BOOL := FALSE;
	END_VAR

	VAR_OUTPUT
		Y :	REAL;
		LIM :	BOOL;
	END_VAR

	VAR
		integ :	INTEGRATE;
		diff :	FT_DERIV;
		YI :	REAL;
	END_VAR

	IF tn = 0.0 OR rst THEN
		integ(E := FALSE, Y := YI);
		YI := integ.Y;
		YI := 0.0;
	ELSE
		integ(X := IN, K := 1.0 / TN, E := NOT LIM, Y := YI);
		YI := integ.Y;
	END_IF;

	(* add up integrator and linear part *)
	Y := KP * (IN + YI);

	(* run differentiator *)
	diff(IN := IN, K := TV);

	(* set lim before differentiator is added to stop integrator if necessary *)
	IF Y > LIM_L AND Y < LIM_H THEN
		LIM := FALSE;
	ELSE
		LIM := TRUE;
	END_IF;

	Y := LIMIT(LIM_L, Y + KP * diff.out, LIM_H);

END_FUNCTION_BLOCK

PROGRAM program0
	VAR
		IN :	REAL;
		KP :	REAL := 1.0;
		TN :	REAL := 1.0;
		TV :	REAL := 1.0;
		LIM_L :	REAL := -1.0E38;
		LIM_H :	REAL := 1.0E38;
		RST :	BOOL := FALSE;

		Y :	REAL;
		LIM :	BOOL;

		func_block : FT_PIDW;
	END_VAR
	func_block.IN := IN;
	func_block.KP := KP;
	func_block.TN := TN;
	func_block.TV := TV;
	func_block.LIM_L := LIM_L;
	func_block.LIM_H := LIM_H;
	func_block.RST := RST;

	func_block();
	Y := func_block.Y;
	LIM := func_block.LIM;
END_PROGRAM

CONFIGURATION Config0

	VAR_GLOBAL
		PLC_TICKS_PER_SEC :	INT;
		PLC_SYS_TICK_CNT :	DINT;
	END_VAR

	RESOURCE Res0 ON PLC
		TASK task0(INTERVAL := T#20ms,PRIORITY := 0);
		PROGRAM instance0 WITH task0 : program0;
	END_RESOURCE

END_CONFIGURATION

(* ---- FT_PIDWL.ST ---- *)
FUNCTION_BLOCK T_PLC_US_Block
	VAR_OUTPUT
		T_PLC_US :	UDINT;
	END_VAR

	VAR_EXTERNAL
		PLC_TICKS_PER_SEC :	INT;
		PLC_SYS_TICK_CNT :	DINT;
	END_VAR

	VAR
		debug :	BOOL;
		N :	INT;
		Offset :	UDINT;
		temp :	DWORD := DWORD#1;
		mode :	BOOL;
		faktor :	UDINT;
		init :	BOOL;
		v_plc_ticks_per_sec :	UDINT;
		base :	UDINT := UDINT#1000000;
	END_VAR

	IF init = FALSE THEN
		v_plc_ticks_per_sec := INT_TO_UDINT(PLC_TICKS_PER_SEC);
		IF v_plc_ticks_per_sec = UDINT#1024 THEN
			faktor := UDINT#1000;
			mode := FALSE;
		ELSIF v_plc_ticks_per_sec > UDINT#0 THEN
			IF v_plc_ticks_per_sec <= base THEN
				faktor := base / v_plc_ticks_per_sec;
				mode := FALSE;
			ELSE
				faktor := v_plc_ticks_per_sec / base;
				mode := TRUE;
			END_IF;
		ELSE
			faktor := UDINT#1;
		END_IF;
		init := TRUE;
	END_IF;

	IF mode THEN
		T_PLC_US := DINT_TO_UDINT(PLC_SYS_TICK_CNT) / faktor;
	ELSE
		T_PLC_US := DINT_TO_UDINT(PLC_SYS_TICK_CNT) * faktor;
	END_IF;

	IF debug THEN
		T_PLC_US := (DWORD_TO_UDINT(SHL(UDINT_TO_DWORD(T_PLC_US),N) OR SHL(temp,N)) - UDINT#1) + Offset;
	END_IF;
END_FUNCTION_BLOCK

FUNCTION_BLOCK FT_PIWL

	VAR_INPUT
		IN :	REAL;
		KP :	REAL := 1.0;
		KI :	REAL := 1.0;
		LIM_L :	REAL := -1.0E38;
		LIM_H :	REAL := 1.0E38;
		RST :	BOOL;
	END_VAR

	VAR_OUTPUT
		Y :	REAL;
		LIM :	BOOL;
	END_VAR

	VAR
		init :	BOOL;
		tx :	UDINT;
		tc :	REAL;
		t_last :	UDINT;
		in_last :	REAL;
		i :	REAL;
		p :	REAL;
		T_PLC_US :	T_PLC_US_Block;
	END_VAR

	IF NOT init OR RST THEN
		init := TRUE;
		in_last := in;
		T_PLC_US();
		t_last := T_PLC_US.T_PLC_US;
		i := 0.0;
		tc := 0.0;
	ELSE
		(* read last cycle time in Microseconds *)
		T_PLC_US();
		tx := T_PLC_US.T_PLC_US;
		tc := UDINT_TO_REAL(tx - t_last);
		t_last := tx;

		(* calculate proportional part *)
		p := KP * IN;

		(* run integrator *)
		i := (IN + in_last) * 5.0E-7 * KI * tc + i;
		in_last := IN;

		(* calculate output Y *)
		Y := p + i;

		(* check output for limits *)
		IF Y >= LIM_H THEN
			Y := LIM_H;
			IF ki <> 0.0 THEN
				i := LIM_H - p;
			ELSE
				i := 0.0;
			END_IF;
			LIM := TRUE;
		ELSIF Y <= LIM_L THEN
			Y := LIM_L;
			IF ki <> 0.0 THEN
				i := LIM_L - p;
			ELSE
				i := 0.0;
			END_IF;
			LIM := TRUE;
		ELSE
			LIM := FALSE;
		END_IF;
	END_IF;
END_FUNCTION_BLOCK

FUNCTION_BLOCK FT_DERIV
	VAR_INPUT
		IN :	REAL;
		K :	REAL := 1.0;
		RUN :	BOOL := TRUE;
	END_VAR

	VAR_OUTPUT
		OUT :	REAL;
	END_VAR

	VAR
		old :	REAL;
		tx :	UDINT;
		last :	UDINT;
		init :	BOOL;
		tc :	REAL;
		T_PLC_US :	T_PLC_US_Block;
	END_VAR

	T_PLC_US();
	tx:= T_PLC_US.T_PLC_US;
	tc := UDINT_TO_REAL(tx - last);

	IF NOT init THEN
		init := TRUE;
		old := in;
	ELSIF run AND tc > 0.0 THEN
		out := (in - old) / tc * 1000000.0 * K;
		old := in;
	ELSE
		out := 0.0;
	END_IF;

	last := tx;

	T_PLC_US();
	tx:= T_PLC_US.T_PLC_US;

	IF NOT init THEN
		init := TRUE;
	ELSIF run AND tx - last > UDINT#0 THEN
		out := (in - old) / UDINT_TO_REAL(tx - last) * 1000000.0 * K;
	ELSE
		out := 0.0;
	END_IF;
	old := in;
	last := tx;
END_FUNCTION_BLOCK

FUNCTION_BLOCK FT_PIDWL
	VAR_INPUT
		IN :	REAL;
		KP :	REAL := 1.0;
		TN :	REAL := 1.0;
		TV :	REAL := 1.0;
		LIM_L :	REAL := -1.0E38;
		LIM_H :	REAL := 1.0E38;
		RST :	BOOL;
	END_VAR

	VAR_OUTPUT
		Y :	REAL;
		LIM :	BOOL;
	END_VAR

	VAR
		piwl :	FT_PIWL;
		diff :	FT_DERIV;
	END_VAR

	IF rst THEN
		piwl(rst := TRUE);
		piwl.RST := FALSE;
	ELSE
		IF TN = 0.0 THEN
			piwl(in := IN * KP, KP := 1.0, KI := 0.0, LIM_L := LIM_L, LIM_H := LIM_H);
		ELSE
			piwl(in := IN * KP, KP := 1.0, KI := 1.0 / TN, LIM_L := LIM_L, LIM_H := LIM_H);
		END_IF;

		diff(IN := IN, K := KP * TV);
		Y := piwl.Y + diff.out;

		IF Y < LIM_L THEN
			LIM := TRUE;
			Y := LIM_L;
		ELSIF Y > LIM_H THEN
			LIM := TRUE;
			Y := LIM_H;
		ELSE
			LIM := FALSE;
		END_IF;
	END_IF;
END_FUNCTION_BLOCK

PROGRAM program0
  VAR
	IN    :	REAL;
	KP    :	REAL;
	TN    :	REAL;
	TV    :	REAL;
	LIM_L :	REAL;
	LIM_H :	REAL;
	RST   :	BOOL;

	Y :	REAL;
	LIM :	BOOL;

	func_block : FT_PIDWL;
  END_VAR
	func_block.IN    :=IN   ;
	func_block.KP    :=KP   ;
	func_block.TN    :=TN   ;
	func_block.TV    :=TV   ;
	func_block.LIM_L :=LIM_L;
	func_block.LIM_H :=LIM_H;
	func_block.RST   :=RST  ;
	func_block();
	Y := func_block.Y;
	LIM := func_block.LIM;
END_PROGRAM

CONFIGURATION Config0
	VAR_GLOBAL
		PLC_TICKS_PER_SEC :	INT;
		PLC_SYS_TICK_CNT :	DINT;
	END_VAR

	RESOURCE Res0 ON PLC
		TASK task0(INTERVAL := T#20ms,PRIORITY := 0);
		PROGRAM instance0 WITH task0 : program0;
	END_RESOURCE
END_CONFIGURATION

(* ---- FT_PIW.ST ---- *)
FUNCTION_BLOCK T_PLC_MS_block
	VAR_OUTPUT
		T_PLC_MS :	UDINT;
	END_VAR

	VAR_EXTERNAL
		PLC_TICKS_PER_SEC :	INT;
		PLC_SYS_TICK_CNT :	DINT;
	END_VAR

	VAR
		debug :	BOOL;(*Debug-Mode ON / OFF*)
		N :	INT;(*Debug-Faktor*)
		Offset :	UDINT;(*Debug-Offset*)
		temp :	DWORD := DWORD#1;(*Debug-Offset*)
		mode :	BOOL;(*modus*)
		faktor :	UDINT;(*Systemtakt-Faktor*)
		init :	BOOL;
		v_plc_ticks_per_sec :	UDINT;
		base :	UDINT := UDINT#1000;
	END_VAR

	IF init = FALSE THEN
		v_plc_ticks_per_sec := INT_TO_UDINT(PLC_TICKS_PER_SEC);
		IF v_plc_ticks_per_sec = UDINT#1024 THEN
			faktor := UDINT#1;
			mode := FALSE;
		ELSIF v_plc_ticks_per_sec > UDINT#0 THEN
			IF v_plc_ticks_per_sec <= base THEN
				faktor := base / v_plc_ticks_per_sec;
				mode := FALSE;
			ELSE
				faktor := v_plc_ticks_per_sec / base;
				mode := TRUE;
			END_IF;
		ELSE
			faktor := UDINT#1;
		END_IF;
		init := TRUE;
	END_IF;

	IF mode THEN
		T_PLC_MS := DINT_TO_UDINT(PLC_SYS_TICK_CNT) / faktor;
	ELSE
		T_PLC_MS := DINT_TO_UDINT(PLC_SYS_TICK_CNT) * faktor;
	END_IF;

	IF debug THEN
		T_PLC_MS := (DWORD_TO_UDINT(SHL(UDINT_TO_DWORD(T_PLC_MS),N) OR SHL(temp,N)) - UDINT#1) + Offset;
	END_IF;
END_FUNCTION_BLOCK

FUNCTION_BLOCK INTEGRATE

	VAR_INPUT
		E :	BOOL := TRUE;
		X :	REAL;
		K :	REAL := 1.0;
	END_VAR

	VAR_IN_OUT
		Y :	REAL;
	END_VAR

	VAR
		X_last :	REAL;
		init :	BOOL;
		T_PLC_MS :	T_PLC_MS_block;
		last :	UDINT;
		tx :	UDINT;
	END_VAR

	T_PLC_MS();
	tx:= T_PLC_MS.T_PLC_MS;

	IF NOT init THEN
		init := TRUE;
		X_last := X;
	ELSIF E THEN
		Y := (X + X_LAST) * 0.5E-3 * UDINT_TO_REAL(tx-last) * K + Y;
		X_last := X;
	END_IF;
	last := tx;

END_FUNCTION_BLOCK

FUNCTION_BLOCK FT_INT_Block

	VAR_INPUT
		IN :	REAL;
		K :	REAL := 1.0;
		RUN :	BOOL := TRUE;
		RST :	BOOL;
		OUT_MIN :	REAL := REAL#-1.0E-37;
		OUT_MAX :	REAL := REAL#1.0E37;
	END_VAR

	VAR_OUTPUT
		OUT :	REAL;
		LIM :	BOOL;
	END_VAR

	VAR
		INTEG :	INTEGRATE;
	END_VAR

	IF rst THEN
		out := 0.0;
	ELSE
		integ(X := IN, E := RUN, K := K, Y := out);
		out := integ.Y;
	END_IF;

	(* limit the outputs *)
	IF out >= OUT_MAX THEN
		out := out_max;
		LIM := TRUE;
	ELSIF out <= out_min THEN
		out := out_min;
		lim := TRUE;
	ELSE
		lim := FALSE;
	END_IF;

END_FUNCTION_BLOCK

FUNCTION_BLOCK FT_PIW

	VAR_INPUT
		IN :	REAL;
		KP :	REAL := 1.0;
		KI :	REAL := 1.0;
		LIM_L :	REAL := -1.0E38;
		LIM_H :	REAL := 1.0E38;
		RST :	BOOL := FALSE;
	END_VAR

	VAR_OUTPUT
		Y :	REAL;
		LIM :	BOOL;
	END_VAR

	VAR
		integ :	FT_INT_Block;
	END_VAR

	integ(IN := IN, K := KI, RUN := NOT LIM, RST := RST);

	(* set output value *)
	Y := KP * IN + integ.Out;

	(* check for limits *)
	IF Y < LIM_L THEN
		Y := LIM_L;
		LIM := TRUE;
	ELSIF Y > LIM_H THEN
		Y := LIM_H;
		LIM := TRUE;
	ELSE
		LIM := FALSE;
	END_IF;

END_FUNCTION_BLOCK

PROGRAM program0
	VAR
		IN :	REAL;
		KP :	REAL := 1.0;
		KI :	REAL := 1.0;
		LIM_L :	REAL := -1.0E38;
		LIM_H :	REAL := 1.0E38;
		RST :	BOOL := FALSE;

		Y :	REAL;
		LIM :	BOOL;

		func_block : FT_PIW;
	END_VAR
	func_block.IN := IN;
	func_block.KP := KP;
	func_block.KI := KI;
	func_block.LIM_L := LIM_L;
	func_block.LIM_H := LIM_H;
	func_block.RST := RST;
	func_block();
	Y := func_block.Y;
	LIM := func_block.LIM;
END_PROGRAM

CONFIGURATION Config0

	VAR_GLOBAL
		PLC_TICKS_PER_SEC :	INT;
		PLC_SYS_TICK_CNT :	DINT;
	END_VAR

	RESOURCE Res0 ON PLC
		TASK task0(INTERVAL := T#20ms,PRIORITY := 0);
		PROGRAM instance0 WITH task0 : program0;
	END_RESOURCE

END_CONFIGURATION

(* ---- FT_PIWL.ST ---- *)
FUNCTION_BLOCK T_PLC_US_Block
	VAR_OUTPUT
		T_PLC_US :	UDINT;
	END_VAR

	VAR_EXTERNAL
		PLC_TICKS_PER_SEC :	INT;
		PLC_SYS_TICK_CNT :	DINT;
	END_VAR

	VAR
		debug :	BOOL;
		N :	INT;
		Offset :	UDINT;
		temp :	DWORD := DWORD#1;
		mode :	BOOL;
		faktor :	UDINT;
		init :	BOOL;
		v_plc_ticks_per_sec :	UDINT;
		base :	UDINT := UDINT#1000000;
	END_VAR

	IF init = FALSE THEN
		v_plc_ticks_per_sec := INT_TO_UDINT(PLC_TICKS_PER_SEC);
		IF v_plc_ticks_per_sec = UDINT#1024 THEN
			faktor := UDINT#1000;
			mode := FALSE;
		ELSIF v_plc_ticks_per_sec > UDINT#0 THEN
			IF v_plc_ticks_per_sec <= base THEN
				faktor := base / v_plc_ticks_per_sec;
				mode := FALSE;
			ELSE
				faktor := v_plc_ticks_per_sec / base;
				mode := TRUE;
			END_IF;
		ELSE
			faktor := UDINT#1;
		END_IF;
		init := TRUE;
	END_IF;

	IF mode THEN
		T_PLC_US := DINT_TO_UDINT(PLC_SYS_TICK_CNT) / faktor;
	ELSE
		T_PLC_US := DINT_TO_UDINT(PLC_SYS_TICK_CNT) * faktor;
	END_IF;

	IF debug THEN
		T_PLC_US := (DWORD_TO_UDINT(SHL(UDINT_TO_DWORD(T_PLC_US),N) OR SHL(temp,N)) - UDINT#1) + Offset;
	END_IF;
END_FUNCTION_BLOCK

FUNCTION_BLOCK FT_PIWL

	VAR_INPUT
		IN :	REAL;
		KP :	REAL := 1.0;
		KI :	REAL := 1.0;
		LIM_L :	REAL := -1.0E38;
		LIM_H :	REAL := 1.0E38;
		RST :	BOOL;
	END_VAR

	VAR_OUTPUT
		Y :	REAL;
		LIM :	BOOL;
	END_VAR

	VAR
		init :	BOOL;
		tx :	UDINT;
		tc :	REAL;
		t_last :	UDINT;
		in_last :	REAL;
		i :	REAL;
		p :	REAL;
		T_PLC_US :	T_PLC_US_Block;
	END_VAR

	IF NOT init OR RST THEN
		init := TRUE;
		in_last := in;
		T_PLC_US();
		t_last := T_PLC_US.T_PLC_US;
		i := 0.0;
		tc := 0.0;
	ELSE
		(* read last cycle time in Microseconds *)
		T_PLC_US();
		tx := T_PLC_US.T_PLC_US;
		tc := UDINT_TO_REAL(tx - t_last);
		t_last := tx;

		(* calculate proportional part *)
		p := KP * IN;

		(* run integrator *)
		i := (IN + in_last) * 5.0E-7 * KI * tc + i;
		in_last := IN;

		(* calculate output Y *)
		Y := p + i;

		(* check output for limits *)
		IF Y >= LIM_H THEN
			Y := LIM_H;
			IF ki <> 0.0 THEN
				i := LIM_H - p;
			ELSE
				i := 0.0;
			END_IF;
			LIM := TRUE;
		ELSIF Y <= LIM_L THEN
			Y := LIM_L;
			IF ki <> 0.0 THEN
				i := LIM_L - p;
			ELSE
				i := 0.0;
			END_IF;
			LIM := TRUE;
		ELSE
			LIM := FALSE;
		END_IF;
	END_IF;
END_FUNCTION_BLOCK

PROGRAM program0
  VAR
	IN    :	REAL;
	KP    :	REAL;
	KI    :	REAL;
	LIM_L :	REAL;
	LIM_H :	REAL;
	RST   :	BOOL;

	Y :	REAL;
	LIM :	BOOL;

	func_block : FT_PIWL;
  END_VAR
	func_block.IN    :=IN   ;
	func_block.KP    :=KP   ;
	func_block.KI    :=KI   ;
	func_block.LIM_L :=LIM_L;
	func_block.LIM_H :=LIM_H;
	func_block.RST   :=RST  ;
	func_block();
	Y := func_block.Y;
	LIM := func_block.LIM;
END_PROGRAM

CONFIGURATION Config0
	VAR_GLOBAL
		PLC_TICKS_PER_SEC :	INT;
		PLC_SYS_TICK_CNT :	DINT;
	END_VAR

	RESOURCE Res0 ON PLC
		TASK task0(INTERVAL := T#20ms,PRIORITY := 0);
		PROGRAM instance0 WITH task0 : program0;
	END_RESOURCE
END_CONFIGURATION

(* ---- FT_PROFILE.ST ---- *)
FUNCTION_BLOCK T_PLC_MS_block
	VAR_OUTPUT
		T_PLC_MS :	UDINT;
	END_VAR

	VAR_EXTERNAL
		PLC_TICKS_PER_SEC :	INT;
		PLC_SYS_TICK_CNT :	DINT;
	END_VAR

	VAR
		debug :	BOOL;(*Debug-Mode ON / OFF*)
		N :	INT;(*Debug-Faktor*)
		Offset :	UDINT;(*Debug-Offset*)
		temp :	DWORD := DWORD#1;(*Debug-Offset*)
		mode :	BOOL;(*modus*)
		faktor :	UDINT;(*Systemtakt-Faktor*)
		init :	BOOL;
		v_plc_ticks_per_sec :	UDINT;
		base :	UDINT := UDINT#1000;
	END_VAR

	IF init = FALSE THEN
		v_plc_ticks_per_sec := INT_TO_UDINT(PLC_TICKS_PER_SEC);
		IF v_plc_ticks_per_sec = UDINT#1024 THEN
			faktor := UDINT#1;
			mode := FALSE;
		ELSIF v_plc_ticks_per_sec > UDINT#0 THEN
			IF v_plc_ticks_per_sec <= base THEN
				faktor := base / v_plc_ticks_per_sec;
				mode := FALSE;
			ELSE
				faktor := v_plc_ticks_per_sec / base;
				mode := TRUE;
			END_IF;
		ELSE
			faktor := UDINT#1;
		END_IF;
		init := TRUE;
	END_IF;

	IF mode THEN
		T_PLC_MS := DINT_TO_UDINT(PLC_SYS_TICK_CNT) / faktor;
	ELSE
		T_PLC_MS := DINT_TO_UDINT(PLC_SYS_TICK_CNT) * faktor;
	END_IF;

	IF debug THEN
		T_PLC_MS := (DWORD_TO_UDINT(SHL(UDINT_TO_DWORD(T_PLC_MS),N) OR SHL(temp,N)) - UDINT#1) + Offset;
	END_IF;
END_FUNCTION_BLOCK

FUNCTION_BLOCK FT_PROFILE

	VAR_INPUT
		K :	REAL := 1.0;
		O :	REAL := 0.0;
		M :	REAL := 1.0;
		E :	BOOL;
		VALUE_0 :	REAL;
		TIME_1 :	TIME;
		VALUE_1 :	REAL;
		TIME_2 :	TIME;
		VALUE_2 :	REAL;
		TIME_3 :	TIME;
		VALUE_3 :	REAL;
		TIME_10 :	TIME;
		VALUE_10 :	REAL;
		TIME_11 :	TIME;
		VALUE_11 :	REAL;
		TIME_12 :	TIME;
		VALUE_12 :	REAL;
		TIME_13 :	TIME;
		VALUE_13 :	REAL;
	END_VAR

	VAR_OUTPUT
		Y :	REAL;
		RUN :	BOOL;
		ET :	TIME;
	END_VAR

	VAR
		tx :	TIME;
		edge :	BOOL;
		state :	INT;
		ta :	TIME;
		tb :	TIME;
		t0 :	TIME;
		temp :	REAL;
		va :	REAL;
		vb :	REAL;
		T_PLC_MS :	T_PLC_MS_block;
	END_VAR

	T_PLC_MS();
	tx:= UDINT_TO_TIME(T_PLC_MS.T_PLC_MS);

	(* determine start condition *)
	IF E AND NOT edge THEN
		RUN := TRUE;
		ET := t#0s;
		t0 := tx;
		ta := tx;
		tb := multime(time_1, M);
		va := value_0;
		vb := value_1;
		temp := value_0;
		state := 1;
	END_IF;
	edge := E;

	(* generate startup profile *)
	IF run THEN
		CASE state OF
			1:	IF tx - ta >= tb THEN
					ta := ta + tb;
					tb := multime(time_2 - time_1, M);
					va := value_1;
					vb := value_2;
					temp := value_1;
					state := 2;
				ELSE
					temp := ((vb - va) * TIME_TO_REAL(tx - ta) / TIME_TO_REAL(tb) + va);
				END_IF;
			2:	IF tx - ta >= tb THEN
					ta := ta + tb;
					tb := multime(time_3 - time_2, M);
					va := value_2;
					vb := value_3;
					temp := value_2;
					state := 3;
				ELSE
					temp := ((vb - va) * TIME_TO_REAL(tx - ta) / TIME_TO_REAL(tb) + va);
				END_IF;
			3:	IF tx - ta >= tb THEN
					ta := ta + tb;
					tb := multime(time_10 - time_3, M);
					va := value_3;
					vb := value_10;
					temp := value_3;
					state := 4;
				ELSE
					temp := ((vb - va) * TIME_TO_REAL(tx - ta) / TIME_TO_REAL(tb) + va);
				END_IF;
			4 :	IF tx - ta >= tb THEN
					ta := ta + tb;
					tb := multime(time_11 - time_10, M);
					va := value_10;
					vb := value_11;
					temp := value_10;
					IF E THEN state := 5; ELSE state := 6; END_IF;
				ELSE
					temp := ((vb - va) * TIME_TO_REAL(tx - ta) / TIME_TO_REAL(tb) + va);
				END_IF;
			5:	(* extend the signal while E is true *)
				IF E THEN
					ta := tx;
				ELSE
					state := 6;
				END_IF;
			6:	IF tx - ta >= tb THEN
					ta := ta + tb;
					tb := multime(time_12 - time_11, M);
					va := value_11;
					vb := value_12;
					temp := value_11;
					state := 7;
				ELSE
					temp := ((vb - va) * TIME_TO_REAL(tx - ta) / TIME_TO_REAL(tb) + va);
				END_IF;
			7:	IF tx - ta >= tb THEN
					ta := ta + tb;
					tb := multime(time_13 - time_12, M);
					va := value_12;
					vb := value_13;
					temp := value_12;
					state := 8;
				ELSE
					temp := ((vb - va) * TIME_TO_REAL(tx - ta) / TIME_TO_REAL(tb) + va);
				END_IF;
			8:	IF tx - ta >= tb THEN
					temp := value_13;
					run := FALSE;
				ELSE
					temp := ((vb - va) * TIME_TO_REAL(tx - ta) / TIME_TO_REAL(tb) + va);
				END_IF;
		END_CASE;
		Y := temp * K + O;
		ET := tx - t0;
	END_IF;

END_FUNCTION_BLOCK

PROGRAM program0
	VAR
		K :	REAL := 1.0;
		O :	REAL := 0.0;
		M :	REAL := 1.0;
		E :	BOOL;
		VALUE_0 :	REAL;
		TIME_1 :	TIME;
		VALUE_1 :	REAL;
		TIME_2 :	TIME;
		VALUE_2 :	REAL;
		TIME_3 :	TIME;
		VALUE_3 :	REAL;
		TIME_10 :	TIME;
		VALUE_10 :	REAL;
		TIME_11 :	TIME;
		VALUE_11 :	REAL;
		TIME_12 :	TIME;
		VALUE_12 :	REAL;
		TIME_13 :	TIME;
		VALUE_13 :	REAL;

		Y :	REAL;
		RUN :	BOOL;
		ET :	TIME;

		func_block : FT_PROFILE;
	END_VAR
	func_block.K  := K ;
	func_block.O  := O ;
	func_block.M  := M ;
	func_block.E  := E ;
	func_block.VALUE_0  := VALUE_0 ;
	func_block.TIME_1  := TIME_1 ;
	func_block.VALUE_1  := VALUE_1 ;
	func_block.TIME_2  := TIME_2 ;
	func_block.VALUE_2  := VALUE_2 ;
	func_block.TIME_3  := TIME_3 ;
	func_block.VALUE_3  := VALUE_3 ;
	func_block.TIME_10  := TIME_10 ;
	func_block.VALUE_10  := VALUE_10 ;
	func_block.TIME_11  := TIME_11 ;
	func_block.VALUE_11  := VALUE_11 ;
	func_block.TIME_12  := TIME_12 ;
	func_block.VALUE_12  := VALUE_12 ;
	func_block.TIME_13  := TIME_13 ;
	func_block.VALUE_13  := VALUE_13 ;
	func_block();
	Y := func_block.Y;
	RUN := func_block.RUN;
	ET := func_block.ET;
END_PROGRAM

CONFIGURATION Config0

	VAR_GLOBAL
		PLC_TICKS_PER_SEC :	INT;
		PLC_SYS_TICK_CNT :	DINT;
	END_VAR

	RESOURCE Res0 ON PLC
		TASK task0(INTERVAL := T#20ms,PRIORITY := 0);
		PROGRAM instance0 WITH task0 : program0;
	END_RESOURCE

END_CONFIGURATION

(* ---- FT_PT1.ST ---- *)
FUNCTION_BLOCK T_PLC_US_Block

	VAR_OUTPUT
		T_PLC_US :	UDINT;
	END_VAR

	VAR_EXTERNAL
		PLC_TICKS_PER_SEC :	INT;
		PLC_SYS_TICK_CNT :	DINT;
	END_VAR

	VAR
		debug :	BOOL;
		N :	INT;
		Offset :	UDINT;
		temp :	DWORD := DWORD#1;
		mode :	BOOL;
		faktor :	UDINT;
		init :	BOOL;
		v_plc_ticks_per_sec :	UDINT;
		base :	UDINT := UDINT#1000000;
	END_VAR

	IF init = FALSE THEN
		v_plc_ticks_per_sec := INT_TO_UDINT(PLC_TICKS_PER_SEC);
		IF v_plc_ticks_per_sec = UDINT#1024 THEN
			faktor := UDINT#1000;
			mode := FALSE;
		ELSIF v_plc_ticks_per_sec > UDINT#0 THEN
			IF v_plc_ticks_per_sec <= base THEN
				faktor := base / v_plc_ticks_per_sec;
				mode := FALSE;
			ELSE
				faktor := v_plc_ticks_per_sec / base;
				mode := TRUE;
			END_IF;
		ELSE
			faktor := UDINT#1;
		END_IF;
		init := TRUE;
	END_IF;

	IF mode THEN
		T_PLC_US := DINT_TO_UDINT(PLC_SYS_TICK_CNT) / faktor;
	ELSE
		T_PLC_US := DINT_TO_UDINT(PLC_SYS_TICK_CNT) * faktor;
	END_IF;

	IF debug THEN
		T_PLC_US := (DWORD_TO_UDINT(SHL(UDINT_TO_DWORD(T_PLC_US),N) OR SHL(temp,N)) - UDINT#1) + Offset;
	END_IF;

END_FUNCTION_BLOCK

FUNCTION_BLOCK FT_PT1

	VAR_INPUT
		IN :	REAL;
		T :	TIME;
		K :	REAL := 1.0;
	END_VAR

	VAR_OUTPUT
		OUT :	REAL;
	END_VAR

	VAR
		last :	UDINT;
		tx :	UDINT;
		init :	BOOL;
		T_PLC_US :	T_PLC_US_Block;
	END_VAR

	T_PLC_US();
	tx:= T_PLC_US.T_PLC_US;

	IF NOT init OR T = t#0s THEN
		init := TRUE;
		out := K * in;
	ELSE
		out := out + (in * K - out) * UDINT_TO_REAL(Tx - last) / TIME_TO_REAL(T) * 1.0E-3;
		IF ABS(out) < 1.0E-20 THEN out := 0.0; END_IF;
	END_IF;
	last := tx;

END_FUNCTION_BLOCK

PROGRAM program0
  VAR
	IN :	REAL;
	T  :	TIME;
	K  :	REAL := 1.0;

	OUT :	REAL;

	func_block : FT_PT1;
  END_VAR
	func_block.IN :=IN;
	func_block.T  :=T ;
	func_block.K  :=K ;
	func_block();
	OUT := func_block.OUT;
END_PROGRAM

CONFIGURATION Config0

	VAR_GLOBAL
		PLC_TICKS_PER_SEC :	INT;
		PLC_SYS_TICK_CNT :	DINT;
	END_VAR

	RESOURCE Res0 ON PLC
		TASK task0(INTERVAL := T#20ms,PRIORITY := 0);
		PROGRAM instance0 WITH task0 : program0;
	END_RESOURCE

END_CONFIGURATION

(* ---- FT_PT2.ST ---- *)
FUNCTION_BLOCK T_PLC_MS_block
	VAR_OUTPUT
		T_PLC_MS :	UDINT;
	END_VAR

	VAR_EXTERNAL
		PLC_TICKS_PER_SEC :	INT;
		PLC_SYS_TICK_CNT :	DINT;
	END_VAR

	VAR
		debug :	BOOL;(*Debug-Mode ON / OFF*)
		N :	INT;(*Debug-Faktor*)
		Offset :	UDINT;(*Debug-Offset*)
		temp :	DWORD := DWORD#1;(*Debug-Offset*)
		mode :	BOOL;(*modus*)
		faktor :	UDINT;(*Systemtakt-Faktor*)
		init :	BOOL;
		v_plc_ticks_per_sec :	UDINT;
		base :	UDINT := UDINT#1000;
	END_VAR

	IF init = FALSE THEN
		v_plc_ticks_per_sec := INT_TO_UDINT(PLC_TICKS_PER_SEC);
		IF v_plc_ticks_per_sec = UDINT#1024 THEN
			faktor := UDINT#1;
			mode := FALSE;
		ELSIF v_plc_ticks_per_sec > UDINT#0 THEN
			IF v_plc_ticks_per_sec <= base THEN
				faktor := base / v_plc_ticks_per_sec;
				mode := FALSE;
			ELSE
				faktor := v_plc_ticks_per_sec / base;
				mode := TRUE;
			END_IF;
		ELSE
			faktor := UDINT#1;
		END_IF;
		init := TRUE;
	END_IF;

	IF mode THEN
		T_PLC_MS := DINT_TO_UDINT(PLC_SYS_TICK_CNT) / faktor;
	ELSE
		T_PLC_MS := DINT_TO_UDINT(PLC_SYS_TICK_CNT) * faktor;
	END_IF;

	IF debug THEN
		T_PLC_MS := (DWORD_TO_UDINT(SHL(UDINT_TO_DWORD(T_PLC_MS),N) OR SHL(temp,N)) - UDINT#1) + Offset;
	END_IF;
END_FUNCTION_BLOCK

FUNCTION_BLOCK INTEGRATE

	VAR_INPUT
		E :	BOOL := TRUE;
		X :	REAL;
		K :	REAL := 1.0;
	END_VAR

	VAR_IN_OUT
		Y :	REAL;
	END_VAR

	VAR
		X_last :	REAL;
		init :	BOOL;
		T_PLC_MS :	T_PLC_MS_block;
		last :	UDINT;
		tx :	UDINT;
	END_VAR

	T_PLC_MS();
	tx:= T_PLC_MS.T_PLC_MS;

	IF NOT init THEN
		init := TRUE;
		X_last := X;
	ELSIF E THEN
		Y := (X + X_LAST) * 0.5E-3 * UDINT_TO_REAL(tx-last) * K + Y;
		X_last := X;
	END_IF;
	last := tx;

END_FUNCTION_BLOCK

FUNCTION_BLOCK FT_PT2

	VAR_INPUT
		IN :	REAL;
		T :	TIME;
		D :	REAL;
		K :	REAL := 1.0;
	END_VAR

	VAR_OUTPUT
		OUT :	REAL;
	END_VAR

	VAR
		init :	BOOL;
		int1 :	INTEGRATE;
		int2 :	INTEGRATE;
		tn :	REAL;
		I1 :	REAL;
		I2 :	REAL;
		tn2 :	REAL;
	END_VAR

	IF NOT init OR T = T#0s THEN
		init := TRUE;
		out := K * in;
		I2 := out;
	ELSE
		TN := TIME_TO_REAL(T) / 1000.0;
		tn2 := TN * TN;
		int1(X := in * K / tn2 - I1 * 0.5 * D / TN - I2 / TN2, Y := I1);
		I1 := int1.Y;
		int2(X := I1,Y := I2);
		I2 := int2.Y;
		out := I2;
	END_IF;

END_FUNCTION_BLOCK

PROGRAM program0
	VAR
		IN :	REAL;
		T :	TIME;
		D :	REAL;
		K :	REAL := 1.0;

		OUT :	REAL;

		func_block : FT_PT2;
	END_VAR
	func_block.IN := IN;
	func_block.T := T;
	func_block.D := D;
	func_block.K := K;
	func_block();
	OUT := func_block.OUT;
END_PROGRAM

CONFIGURATION Config0

	VAR_GLOBAL
		PLC_TICKS_PER_SEC :	INT;
		PLC_SYS_TICK_CNT :	DINT;
	END_VAR

	RESOURCE Res0 ON PLC
		TASK task0(INTERVAL := T#20ms,PRIORITY := 0);
		PROGRAM instance0 WITH task0 : program0;
	END_RESOURCE

END_CONFIGURATION

(* ---- FT_RMP.ST ---- *)
FUNCTION_BLOCK T_PLC_MS_block
	VAR_OUTPUT
		T_PLC_MS :	UDINT;
	END_VAR

	VAR_EXTERNAL
		PLC_TICKS_PER_SEC :	INT;
		PLC_SYS_TICK_CNT :	DINT;
	END_VAR

	VAR
		debug :	BOOL;(*Debug-Mode ON / OFF*)
		N :	INT;(*Debug-Faktor*)
		Offset :	UDINT;(*Debug-Offset*)
		temp :	DWORD := DWORD#1;(*Debug-Offset*)
		mode :	BOOL;(*modus*)
		faktor :	UDINT;(*Systemtakt-Faktor*)
		init :	BOOL;
		v_plc_ticks_per_sec :	UDINT;
		base :	UDINT := UDINT#1000;
	END_VAR

	IF init = FALSE THEN
		v_plc_ticks_per_sec := INT_TO_UDINT(PLC_TICKS_PER_SEC);
		IF v_plc_ticks_per_sec = UDINT#1024 THEN
			faktor := UDINT#1;
			mode := FALSE;
		ELSIF v_plc_ticks_per_sec > UDINT#0 THEN
			IF v_plc_ticks_per_sec <= base THEN
				faktor := base / v_plc_ticks_per_sec;
				mode := FALSE;
			ELSE
				faktor := v_plc_ticks_per_sec / base;
				mode := TRUE;
			END_IF;
		ELSE
			faktor := UDINT#1;
		END_IF;
		init := TRUE;
	END_IF;

	IF mode THEN
		T_PLC_MS := DINT_TO_UDINT(PLC_SYS_TICK_CNT) / faktor;
	ELSE
		T_PLC_MS := DINT_TO_UDINT(PLC_SYS_TICK_CNT) * faktor;
	END_IF;

	IF debug THEN
		T_PLC_MS := (DWORD_TO_UDINT(SHL(UDINT_TO_DWORD(T_PLC_MS),N) OR SHL(temp,N)) - UDINT#1) + Offset;
	END_IF;
END_FUNCTION_BLOCK

FUNCTION_BLOCK FT_RMP

	VAR_INPUT
		RMP :	BOOL := TRUE;
		IN :	REAL;
		KR :	REAL;
		KF :	REAL;
	END_VAR

	VAR_OUTPUT
		OUT :	REAL;
		BUSY :	BOOL;
		UD :	BOOL;
	END_VAR

	VAR
		tx :	TIME;
		last :	TIME;
		init :	BOOL;
		T_PLC_MS :	T_PLC_MS_block;
	END_VAR

	T_PLC_MS();
	tx:= UDINT_TO_TIME(T_PLC_MS.T_PLC_MS) - last;

	IF NOT init THEN
		init := TRUE;
		last := tx;
		tx := t#0s;
		out := in;
	END_IF;
	IF NOT rmp THEN
		out := in;
		busy := FALSE;
	ELSIF out > in THEN
		(* ramp down *)
		out := out - TIME_TO_REAL(tx) * 0.001 * KF;
		out := MAX(in, out);
	ELSIF out < in THEN
		(* ramp up *)
		out := out + TIME_TO_REAL(tx) * 0.001 * KR;
		out := MIN(in, out);
	END_IF;

	(* set busy and dir flags *)
	IF out < in THEN
		busy := TRUE;
		ud := TRUE;
	ELSIF out > in THEN
		busy := TRUE;
		ud := FALSE;
	ELSE
		busy := FALSE;
	END_IF;
	last := last + tx;

END_FUNCTION_BLOCK

PROGRAM program0
	VAR
		RMP :	BOOL := TRUE;
		IN :	REAL;
		KR :	REAL;
		KF :	REAL;

		OUT :	REAL;
		BUSY :	BOOL;
		UD :	BOOL;

		func_block : FT_RMP;
	END_VAR
	func_block.RMP := RMP;
	func_block.IN := IN;
	func_block.KR := KR;
	func_block.KF := KF;
	func_block();
	OUT := func_block.OUT;
	BUSY := func_block.BUSY;
	UD := func_block.UD;

END_PROGRAM

CONFIGURATION Config0

	VAR_GLOBAL
		PLC_TICKS_PER_SEC :	INT;
		PLC_SYS_TICK_CNT :	DINT;
	END_VAR

	RESOURCE Res0 ON PLC
		TASK task0(INTERVAL := T#20ms,PRIORITY := 0);
		PROGRAM instance0 WITH task0 : program0;
	END_RESOURCE

END_CONFIGURATION

(* ---- FT_TN16.ST ---- *)
TYPE
  	oscat_arr_0_15               : ARRAY [0..15]    OF REAL;
END_TYPE

FUNCTION_BLOCK T_PLC_MS_Block
	VAR_OUTPUT
		T_PLC_MS :	UDINT;
	END_VAR

	VAR_EXTERNAL
		PLC_TICKS_PER_SEC :	INT;
		PLC_SYS_TICK_CNT :	DINT;
	END_VAR

	VAR
		debug :	BOOL;(*Debug-Mode ON / OFF*)
		N :	INT;(*Debug-Faktor*)
		Offset :	UDINT;(*Debug-Offset*)
		temp :	DWORD := DWORD#1;(*Debug-Offset*)
		mode :	BOOL;(*modus*)
		faktor :	UDINT;(*Systemtakt-Faktor*)
		init :	BOOL;
		v_plc_ticks_per_sec :	UDINT;
		base :	UDINT := UDINT#1000;
	END_VAR

	IF init = FALSE THEN
		v_plc_ticks_per_sec := INT_TO_UDINT(PLC_TICKS_PER_SEC);
		IF v_plc_ticks_per_sec = UDINT#1024 THEN
			faktor := UDINT#1;
			mode := FALSE;
		ELSIF v_plc_ticks_per_sec > UDINT#0 THEN
			IF v_plc_ticks_per_sec <= base THEN
				faktor := base / v_plc_ticks_per_sec;
				mode := FALSE;
			ELSE
				faktor := v_plc_ticks_per_sec / base;
				mode := TRUE;
			END_IF;
		ELSE
			faktor := UDINT#1;
		END_IF;
		init := TRUE;
	END_IF;

	IF mode THEN
		T_PLC_MS := DINT_TO_UDINT(PLC_SYS_TICK_CNT) / faktor;
	ELSE
		T_PLC_MS := DINT_TO_UDINT(PLC_SYS_TICK_CNT) * faktor;
	END_IF;

	IF debug THEN
		T_PLC_MS := (DWORD_TO_UDINT(SHL(UDINT_TO_DWORD(T_PLC_MS),N) OR SHL(temp,N)) - UDINT#1) + Offset;
	END_IF;
END_FUNCTION_BLOCK

FUNCTION_BLOCK FT_TN16
	VAR_INPUT
		IN :	REAL;
		T :	TIME;
	END_VAR

	VAR_OUTPUT
		OUT :	REAL;
		TRIG :	BOOL;
	END_VAR

	VAR
		length :	INT := 16;
		X :	oscat_arr_0_15;
		cnt :	INT;
		last :	TIME;
		tx :	TIME;
		init :	BOOL;
		T_PLC_MS :	T_PLC_MS_Block;
	END_VAR

	T_PLC_MS();
	tx:= UDINT_TO_TIME(T_PLC_MS.T_PLC_MS);

	trig := FALSE;
	IF NOT init THEN
		x[cnt] := in;
		init := TRUE;
		last := tx;
	ELSIF tx - last >= T / length THEN
		IF cnt = length - 1 THEN cnt := 0; ELSE cnt := cnt + 1; END_IF;
		Out := X[cnt];
		x[cnt] := in;
		last := tx;
		Trig := TRUE;
	END_IF;

END_FUNCTION_BLOCK

PROGRAM program0
  VAR
	IN :	REAL;
	T :	TIME;

	OUT :	REAL;
	TRIG :	BOOL;

	func_block : FT_TN16;
  END_VAR
	func_block.IN  :=IN ;
	func_block.T  :=T ;
	func_block();
	OUT := func_block.OUT;
	TRIG := func_block.TRIG;
END_PROGRAM

CONFIGURATION Config0

	VAR_GLOBAL
		PLC_TICKS_PER_SEC :	INT;
		PLC_SYS_TICK_CNT :	DINT;
	END_VAR

	RESOURCE Res0 ON PLC
		TASK task0(INTERVAL := T#20ms,PRIORITY := 0);
		PROGRAM instance0 WITH task0 : program0;
	END_RESOURCE

END_CONFIGURATION

(* ---- FT_TN64.ST ---- *)
TYPE
	oscat_FT_TN64_array         : ARRAY [0..63]   OF REAL;
END_TYPE

FUNCTION_BLOCK T_PLC_MS_Block
	VAR_OUTPUT
		T_PLC_MS :	UDINT;
	END_VAR

	VAR_EXTERNAL
		PLC_TICKS_PER_SEC :	INT;
		PLC_SYS_TICK_CNT :	DINT;
	END_VAR

	VAR
		debug :	BOOL;(*Debug-Mode ON / OFF*)
		N :	INT;(*Debug-Faktor*)
		Offset :	UDINT;(*Debug-Offset*)
		temp :	DWORD := DWORD#1;(*Debug-Offset*)
		mode :	BOOL;(*modus*)
		faktor :	UDINT;(*Systemtakt-Faktor*)
		init :	BOOL;
		v_plc_ticks_per_sec :	UDINT;
		base :	UDINT := UDINT#1000;
	END_VAR

	IF init = FALSE THEN
		v_plc_ticks_per_sec := INT_TO_UDINT(PLC_TICKS_PER_SEC);
		IF v_plc_ticks_per_sec = UDINT#1024 THEN
			faktor := UDINT#1;
			mode := FALSE;
		ELSIF v_plc_ticks_per_sec > UDINT#0 THEN
			IF v_plc_ticks_per_sec <= base THEN
				faktor := base / v_plc_ticks_per_sec;
				mode := FALSE;
			ELSE
				faktor := v_plc_ticks_per_sec / base;
				mode := TRUE;
			END_IF;
		ELSE
			faktor := UDINT#1;
		END_IF;
		init := TRUE;
	END_IF;

	IF mode THEN
		T_PLC_MS := DINT_TO_UDINT(PLC_SYS_TICK_CNT) / faktor;
	ELSE
		T_PLC_MS := DINT_TO_UDINT(PLC_SYS_TICK_CNT) * faktor;
	END_IF;

	IF debug THEN
		T_PLC_MS := (DWORD_TO_UDINT(SHL(UDINT_TO_DWORD(T_PLC_MS),N) OR SHL(temp,N)) - UDINT#1) + Offset;
	END_IF;
END_FUNCTION_BLOCK

FUNCTION_BLOCK FT_TN64

	VAR_INPUT
		IN :	REAL;
		_T :	TIME;
	END_VAR

	VAR_OUTPUT
		OUT :	REAL;
		TRIG :	BOOL;
	END_VAR

	VAR
		length :	INT := 64;
		X :	oscat_FT_TN64_array;
		cnt :	INT;
		last :	TIME;
		tx :	TIME;
		init :	BOOL;
		T_PLC_MS :	T_PLC_MS_Block;
	END_VAR

	T_PLC_MS();
	tx:= UDINT_TO_TIME(T_PLC_MS.T_PLC_MS);

	trig := FALSE;
	IF NOT init THEN
		x[cnt] := in;
		init := TRUE;
		last := tx;
	ELSIF tx - last >= (_T / length) THEN
		IF cnt = length - 1 THEN cnt := 0; ELSE cnt := cnt + 1; END_IF;
		Out := X[cnt];
		x[cnt] := in;
		last := tx;
		trig := TRUE;
	END_IF;

END_FUNCTION_BLOCK

PROGRAM program0
  VAR
	IN :	REAL;
	_T :	TIME;

	OUT :	REAL;
	TRIG :	BOOL;

	func_block : FT_TN64;
  END_VAR
	func_block.IN  :=IN ;
	func_block._T  :=_T ;
	func_block();
	OUT := func_block.OUT;
	TRIG := func_block.TRIG;
END_PROGRAM

CONFIGURATION Config0

	VAR_GLOBAL
		PLC_TICKS_PER_SEC :	INT;
		PLC_SYS_TICK_CNT :	DINT;
	END_VAR

	RESOURCE Res0 ON PLC
		TASK task0(INTERVAL := T#20ms,PRIORITY := 0);
		PROGRAM instance0 WITH task0 : program0;
	END_RESOURCE

END_CONFIGURATION

(* ---- FT_TN8.ST ---- *)
TYPE
  	oscat_arr_0_7               : ARRAY [0..7]    OF REAL;
END_TYPE

FUNCTION_BLOCK T_PLC_MS_Block
	VAR_OUTPUT
		T_PLC_MS :	UDINT;
	END_VAR

	VAR_EXTERNAL
		PLC_TICKS_PER_SEC :	INT;
		PLC_SYS_TICK_CNT :	DINT;
	END_VAR

	VAR
		debug :	BOOL;(*Debug-Mode ON / OFF*)
		N :	INT;(*Debug-Faktor*)
		Offset :	UDINT;(*Debug-Offset*)
		temp :	DWORD := DWORD#1;(*Debug-Offset*)
		mode :	BOOL;(*modus*)
		faktor :	UDINT;(*Systemtakt-Faktor*)
		init :	BOOL;
		v_plc_ticks_per_sec :	UDINT;
		base :	UDINT := UDINT#1000;
	END_VAR

	IF init = FALSE THEN
		v_plc_ticks_per_sec := INT_TO_UDINT(PLC_TICKS_PER_SEC);
		IF v_plc_ticks_per_sec = UDINT#1024 THEN
			faktor := UDINT#1;
			mode := FALSE;
		ELSIF v_plc_ticks_per_sec > UDINT#0 THEN
			IF v_plc_ticks_per_sec <= base THEN
				faktor := base / v_plc_ticks_per_sec;
				mode := FALSE;
			ELSE
				faktor := v_plc_ticks_per_sec / base;
				mode := TRUE;
			END_IF;
		ELSE
			faktor := UDINT#1;
		END_IF;
		init := TRUE;
	END_IF;

	IF mode THEN
		T_PLC_MS := DINT_TO_UDINT(PLC_SYS_TICK_CNT) / faktor;
	ELSE
		T_PLC_MS := DINT_TO_UDINT(PLC_SYS_TICK_CNT) * faktor;
	END_IF;

	IF debug THEN
		T_PLC_MS := (DWORD_TO_UDINT(SHL(UDINT_TO_DWORD(T_PLC_MS),N) OR SHL(temp,N)) - UDINT#1) + Offset;
	END_IF;
END_FUNCTION_BLOCK

FUNCTION_BLOCK FT_TN8

	VAR_INPUT
		IN :	REAL;
		T :	TIME;
	END_VAR

	VAR_OUTPUT
		OUT :	REAL;
		TRIG :	BOOL;
	END_VAR

	VAR
		length :	INT := 8;
		X :	oscat_arr_0_7;
		cnt :	INT;
		last :	TIME;
		tx :	TIME;
		init :	BOOL;
		T_PLC_MS :	T_PLC_MS_Block;
	END_VAR

	T_PLC_MS();
	tx:= UDINT_TO_TIME(T_PLC_MS.T_PLC_MS);

	trig := FALSE;
	IF NOT init THEN
		x[cnt] := in;
		init := TRUE;
		last := tx;
	ELSIF tx - last >= (T / length) THEN
		IF cnt = length - 1 THEN cnt := 0; ELSE cnt := cnt + 1; END_IF;
		Out := X[cnt];
		x[cnt] := in;
		last := tx;
		trig := TRUE;
	END_IF;

END_FUNCTION_BLOCK

PROGRAM program0
  VAR
	IN :	REAL;
	T :	TIME;

	OUT :	REAL;
	TRIG :	BOOL;

	func_block : FT_TN8;
  END_VAR
	func_block.IN  :=IN ;
	func_block.T  :=T ;
	func_block();
	OUT := func_block.OUT;
	TRIG := func_block.TRIG;
END_PROGRAM

CONFIGURATION Config0

	VAR_GLOBAL
		PLC_TICKS_PER_SEC :	INT;
		PLC_SYS_TICK_CNT :	DINT;
	END_VAR

	RESOURCE Res0 ON PLC
		TASK task0(INTERVAL := T#20ms,PRIORITY := 0);
		PROGRAM instance0 WITH task0 : program0;
	END_RESOURCE

END_CONFIGURATION

(* ---- GEN_BIT.ST ---- *)
FUNCTION BIT_OF_DWORD : BOOL
  VAR_INPUT
    IN : DWORD;
    N : INT;
  END_VAR

  BIT_OF_DWORD := (SHR(in,N) AND 16#00000001) > 0;
END_FUNCTION

FUNCTION_BLOCK GEN_BIT_Block

	VAR_INPUT
		IN0 :	DWORD;
		IN1 :	DWORD;
		IN2 :	DWORD;
		IN3 :	DWORD;
		CLK :	BOOL;
		STEPS :	INT;
		REP :	INT;
		RST :	BOOL;
	END_VAR

	VAR_OUTPUT
		Q0 :	BOOL;
		Q1 :	BOOL;
		Q2 :	BOOL;
		Q3 :	BOOL;
		CNT :	INT;
		RUN :	BOOL;
	END_VAR

	VAR
		r0 :	DWORD;
		r1 :	DWORD;
		r2 :	DWORD;
		r3 :	DWORD;
		rx :	INT := 1;
	END_VAR

	IF clk AND NOT rst THEN
		run := (rep = 0) OR (rx <= rep);
		IF run THEN
			IF cnt = steps THEN
				cnt := 0;
			END_IF;

			IF cnt = 0 THEN
				r0 := in0;
				r1 := in1;
				r2 := in2;
				r3 := in3;
			END_IF;

			IF (cnt < steps) THEN
				Q0 := BIT_OF_DWORD(r0,0);
				Q1 := BIT_OF_DWORD(r1,0);
				Q2 := BIT_OF_DWORD(r2,0);
				Q3 := BIT_OF_DWORD(r3,0);
				r0 := SHR(r0,1);
				r1 := SHR(r1,1);
				r2 := SHR(r2,1);
				r3 := SHR(r3,1);
			END_IF;

			cnt := cnt +1;
			IF (cnt = steps) AND (rep <> 0) THEN rx := rx +1; END_IF;
			IF (rx > rep) AND (rep <> 0) THEN run := FALSE; END_IF;
		END_IF;
	ELSE
		IF rst THEN
			run := FALSE;
			Q0 := FALSE;
			Q1 := FALSE;
			Q2 := FALSE;
			Q3 := FALSE;
			r0 := DWORD#0;
			r1 := DWORD#0;
			r2 := DWORD#0;
			r3 := DWORD#0;
			cnt := 0;
			rx := 1;
		END_IF;
	END_IF;

END_FUNCTION_BLOCK

PROGRAM program0
  VAR
	IN0 :	DWORD;
	IN1 :	DWORD;
	IN2 :	DWORD;
	IN3 :	DWORD;
	CLK :	BOOL;
	STEPS :	INT;
	REP :	INT;
	RST :	BOOL;
	Q0 :	BOOL;
	Q1 :	BOOL;
	Q2 :	BOOL;
	Q3 :	BOOL;
	CNT :	INT;
	RUN :	BOOL;
	func_block : GEN_BIT_Block;
  END_VAR
	func_block.IN0  :=IN0;
	func_block.IN1  :=IN1;
	func_block.IN2  :=IN2;
	func_block.IN3  :=IN3;
	func_block.CLK  :=CLK;
	func_block.STEPS  :=STEPS;
	func_block.REP  :=REP;
	func_block.RST  :=RST;
	func_block();
	Q0 := func_block.Q0;
	Q1 := func_block.Q1;
	Q2 := func_block.Q2;
	Q3 := func_block.Q3;
	CNT := func_block.CNT;
	RUN := func_block.RUN;

END_PROGRAM

CONFIGURATION Config0
	RESOURCE Res0 ON PLC
		TASK task0(INTERVAL := T#20ms,PRIORITY := 0);
		PROGRAM instance0 WITH task0 : program0;
	END_RESOURCE
END_CONFIGURATION

(* ---- GEN_PULSE.ST ---- *)
FUNCTION UDINT_TO_TIME2:TIME

	VAR_INPUT
		IN :	UDINT;
	END_VAR

	UDINT_TO_TIME2 := DINT_TO_TIME(UDINT_TO_DINT(IN));

END_FUNCTION

FUNCTION_BLOCK T_PLC_MS_block
	VAR_OUTPUT
		T_PLC_MS :	UDINT;
	END_VAR

	VAR_EXTERNAL
		PLC_TICKS_PER_SEC :	INT;
		PLC_SYS_TICK_CNT :	DINT;
	END_VAR

	VAR
		debug :	BOOL;(*Debug-Mode ON / OFF*)
		N :	INT;(*Debug-Faktor*)
		Offset :	UDINT;(*Debug-Offset*)
		temp :	DWORD := DWORD#1;(*Debug-Offset*)
		mode :	BOOL;(*modus*)
		faktor :	UDINT;(*Systemtakt-Faktor*)
		init :	BOOL;
		v_plc_ticks_per_sec :	UDINT;
		base :	UDINT := UDINT#1000;
	END_VAR

	IF init = FALSE THEN
		v_plc_ticks_per_sec := INT_TO_UDINT(PLC_TICKS_PER_SEC);
		IF v_plc_ticks_per_sec = UDINT#1024 THEN
			faktor := UDINT#1;
			mode := FALSE;
		ELSIF v_plc_ticks_per_sec > UDINT#0 THEN
			IF v_plc_ticks_per_sec <= base THEN
				faktor := base / v_plc_ticks_per_sec;
				mode := FALSE;
			ELSE
				faktor := v_plc_ticks_per_sec / base;
				mode := TRUE;
			END_IF;
		ELSE
			faktor := UDINT#1;
		END_IF;
		init := TRUE;
	END_IF;

	IF mode THEN
		T_PLC_MS := DINT_TO_UDINT(PLC_SYS_TICK_CNT) / faktor;
	ELSE
		T_PLC_MS := DINT_TO_UDINT(PLC_SYS_TICK_CNT) * faktor;
	END_IF;

	IF debug THEN
		T_PLC_MS := (DWORD_TO_UDINT(SHL(UDINT_TO_DWORD(T_PLC_MS),N) OR SHL(temp,N)) - UDINT#1) + Offset;
	END_IF;

END_FUNCTION_BLOCK

FUNCTION_BLOCK GEN_PULSE_Block

	VAR_INPUT
		ENQ :	BOOL := TRUE;
		PTH :	TIME;
		PTL :	TIME;
	END_VAR

	VAR_OUTPUT
		Q :	BOOL;
	END_VAR

	VAR
		T_PLC_MS :	T_PLC_MS_block;
		tx :	TIME;
		tn :	TIME;
		init :	BOOL;
	END_VAR

	IF enq THEN
		T_PLC_MS();
		tx:= UDINT_TO_TIME(T_PLC_MS.T_PLC_MS);
		IF NOT init THEN init := TRUE; tn := tx; END_IF;
		IF tx - tn >= SEL(Q, PTL, PTH) THEN
			tn := tn + SEL(Q, PTL, PTH);
			Q := NOT Q;
		END_IF;
	ELSE
		Q := FALSE;
		init := FALSE;
	END_IF;

END_FUNCTION_BLOCK

PROGRAM program0
  VAR
	ENQ :	BOOL := TRUE;
	PTH :	TIME;
	PTL :	TIME;
	Q :	BOOL;
	func_block : GEN_PULSE_Block;
  END_VAR
	func_block.ENQ  :=ENQ;
	func_block.PTH  :=PTH;
	func_block.PTL  :=PTL;
	func_block();
	Q := func_block.Q;

END_PROGRAM

CONFIGURATION Config0
	VAR_GLOBAL
		PLC_TICKS_PER_SEC :	INT;
		PLC_SYS_TICK_CNT :	DINT;
	END_VAR
	RESOURCE Res0 ON PLC
		TASK task0(INTERVAL := T#20ms,PRIORITY := 0);
		PROGRAM instance0 WITH task0 : program0;
	END_RESOURCE
END_CONFIGURATION

(* ---- GEN_PW2.ST ---- *)
FUNCTION UDINT_TO_TIME2:TIME

	VAR_INPUT
		IN :	UDINT;
	END_VAR

	UDINT_TO_TIME2 := DINT_TO_TIME(UDINT_TO_DINT(IN));

END_FUNCTION

FUNCTION_BLOCK T_PLC_MS_block
	VAR_OUTPUT
		T_PLC_MS :	UDINT;
	END_VAR

	VAR_EXTERNAL
		PLC_TICKS_PER_SEC :	INT;
		PLC_SYS_TICK_CNT :	DINT;
	END_VAR

	VAR
		debug :	BOOL;
		N :	INT;
		Offset :	UDINT;
		temp :	DWORD := DWORD#1;
		mode :	BOOL;
		faktor :	UDINT;
		init :	BOOL;
		v_plc_ticks_per_sec :	UDINT;
		base :	UDINT := UDINT#1000;
	END_VAR

	IF init = FALSE THEN
		v_plc_ticks_per_sec := INT_TO_UDINT(PLC_TICKS_PER_SEC);
		IF v_plc_ticks_per_sec = UDINT#1024 THEN
			faktor := UDINT#1;
			mode := FALSE;
		ELSIF v_plc_ticks_per_sec > UDINT#0 THEN
			IF v_plc_ticks_per_sec <= base THEN
				faktor := base / v_plc_ticks_per_sec;
				mode := FALSE;
			ELSE
				faktor := v_plc_ticks_per_sec / base;
				mode := TRUE;
			END_IF;
		ELSE
			faktor := UDINT#1;
		END_IF;
		init := TRUE;
	END_IF;

	IF mode THEN
		T_PLC_MS := DINT_TO_UDINT(PLC_SYS_TICK_CNT) / faktor;
	ELSE
		T_PLC_MS := DINT_TO_UDINT(PLC_SYS_TICK_CNT) * faktor;
	END_IF;

	IF debug THEN
		T_PLC_MS := (DWORD_TO_UDINT(SHL(UDINT_TO_DWORD(T_PLC_MS),N) OR SHL(temp,N)) - UDINT#1) + Offset;
	END_IF;

END_FUNCTION_BLOCK

FUNCTION_BLOCK GEN_PW2_Block

	VAR_INPUT
		ENQ :	BOOL;
		TH1 :	TIME;
		TL1 :	TIME;
		TH2 :	TIME;
		TL2 :	TIME;
		TS :	BOOL;
	END_VAR

	VAR_OUTPUT
		Q :	BOOL;
		TH :	TIME;
		TL :	TIME;
	END_VAR

	VAR
		T_PLC_MS :	T_PLC_MS_Block;
		t_high :	TIME;
		t_low :	TIME;
		tx :	TIME;
		start :	TIME;
		init :	BOOL;
		et :	TIME;
	END_VAR

	T_PLC_MS();
	tx:= UDINT_TO_TIME(T_PLC_MS.T_PLC_MS);

	IF NOT init THEN
		start := tx;
		init := TRUE;
		TH := T#0s;
		TL := T#0s;
	END_IF;

	IF TS THEN
		t_high := TH2;
		t_low := TL2;
	ELSE
		t_high := TH1;
		t_low := TL1;
	END_IF;

	IF ENQ THEN
		et := tx - start;
		IF NOT Q THEN
			IF et >= t_low THEN
				Q := TRUE;
				start := tx;
				TL := T#0s;
			ELSE
				TL := et;
			END_IF;
		ELSE
			IF et >= t_high THEN
				Q := FALSE;
				start := tx;
				TH := T#0s;
			ELSE
				TH := et;
			END_IF;
		END_IF;
	ELSE
		Q := FALSE;
		TH := T#0s;
		TL := T#0s;
		start := tx;
	END_IF;

END_FUNCTION_BLOCK

PROGRAM program0
  VAR
	ENQ :	BOOL;
	TH1 :	TIME;
	TL1 :	TIME;
	TH2 :	TIME;
	TL2 :	TIME;
	TS :	BOOL;
	Q :	BOOL;
	TH :	TIME;
	TL :	TIME;
	func_block : GEN_PW2_Block;
  END_VAR
	func_block.ENQ  :=ENQ;
	func_block.TH1  :=TH1;
	func_block.TL1  :=TL1;
	func_block.TH2  :=TH2;
	func_block.TL2  :=TL2;
	func_block.TS  :=TS;
	func_block.TS  :=TS;
	func_block();
	Q := func_block.Q;
	TH := func_block.TH;
	TL := func_block.TL;

END_PROGRAM

CONFIGURATION Config0
	VAR_GLOBAL
		PLC_TICKS_PER_SEC :	INT;
		PLC_SYS_TICK_CNT :	DINT;
	END_VAR
	RESOURCE Res0 ON PLC
		TASK task0(INTERVAL := T#20ms,PRIORITY := 0);
		PROGRAM instance0 WITH task0 : program0;
	END_RESOURCE
END_CONFIGURATION

(* ---- GEN_RDM.ST ---- *)
FUNCTION D_TRUNC : DINT
  VAR_INPUT
    x : REAL;
  END_VAR

  D_TRUNC := REAL_TO_DINT(X);
  IF X > 0.0 THEN
  	IF DINT_TO_REAL(D_TRUNC) > X THEN D_TRUNC := D_TRUNC - DINT#1; END_IF;
  ELSE
  	IF DINT_TO_REAL(D_TRUNC) < X THEN D_TRUNC := D_TRUNC + DINT#1; END_IF;
  END_IF;
END_FUNCTION

FUNCTION BIT_COUNT:INT

	VAR_INPUT
		IN :	DWORD;
	END_VAR

	VAR
		in_temp :	DWORD;
	END_VAR

	in_temp := IN;
	WHILE in_temp > DWORD#0 DO
		IF (in_temp AND DWORD#16#00000001) > DWORD#0 THEN Bit_Count := Bit_Count +1; END_IF;
		in_temp := SHR(in_temp,1);
	END_WHILE;

END_FUNCTION

FUNCTION FRACT:REAL
	VAR_INPUT
		X :	REAL;
	END_VAR

	IF ABS(x) < 2.0E9 THEN
		FRACT := x - DINT_TO_REAL(D_TRUNC(x));
	ELSE
		FRACT := 0.0;
	END_IF;

END_FUNCTION

FUNCTION_BLOCK T_PLC_MS_block
	VAR_OUTPUT
		T_PLC_MS :	UDINT;
	END_VAR

	VAR_EXTERNAL
		PLC_TICKS_PER_SEC :	INT;
		PLC_SYS_TICK_CNT :	DINT;
	END_VAR

	VAR
		debug :	BOOL;(*Debug-Mode ON / OFF*)
		N :	INT;(*Debug-Faktor*)
		Offset :	UDINT;(*Debug-Offset*)
		temp :	DWORD := DWORD#1;(*Debug-Offset*)
		mode :	BOOL;(*modus*)
		faktor :	UDINT;(*Systemtakt-Faktor*)
		init :	BOOL;
		v_plc_ticks_per_sec :	UDINT;
		base :	UDINT := UDINT#1000;
	END_VAR

	IF init = FALSE THEN
		v_plc_ticks_per_sec := INT_TO_UDINT(PLC_TICKS_PER_SEC);
		IF v_plc_ticks_per_sec = UDINT#1024 THEN
			faktor := UDINT#1;
			mode := FALSE;
		ELSIF v_plc_ticks_per_sec > UDINT#0 THEN
			IF v_plc_ticks_per_sec <= base THEN
				faktor := base / v_plc_ticks_per_sec;
				mode := FALSE;
			ELSE
				faktor := v_plc_ticks_per_sec / base;
				mode := TRUE;
			END_IF;
		ELSE
			faktor := UDINT#1;
		END_IF;
		init := TRUE;
	END_IF;

	IF mode THEN
		T_PLC_MS := DINT_TO_UDINT(PLC_SYS_TICK_CNT) / faktor;
	ELSE
		T_PLC_MS := DINT_TO_UDINT(PLC_SYS_TICK_CNT) * faktor;
	END_IF;

	IF debug THEN
		T_PLC_MS := (DWORD_TO_UDINT(SHL(UDINT_TO_DWORD(T_PLC_MS),N) OR SHL(temp,N)) - UDINT#1) + Offset;
	END_IF;

END_FUNCTION_BLOCK

FUNCTION BIT_LOAD_DW:DWORD

	VAR_INPUT
		IN :	DWORD;
		VAL :	BOOL;
		POS :	INT;
	END_VAR

	IF val THEN
		BIT_LOAD_DW := in OR SHL(DWORD#1,pos);
	ELSE
		BIT_LOAD_DW := in AND (NOT SHL(DWORD#1,pos));
	END_IF;

END_FUNCTION

FUNCTION BIT_OF_DWORD : BOOL
  VAR_INPUT
    IN : DWORD;
    N : INT;
  END_VAR

  BIT_OF_DWORD := (SHR(in,N) AND 16#00000001) > 0;
  (* from OSCAT library; www.oscat.de  *)
END_FUNCTION

FUNCTION _INT_TO_UDINT:UDINT
	VAR_INPUT
		IN :	INT;
	END_VAR

	_INT_TO_UDINT := DINT_TO_UDINT(INT_TO_DINT(IN));
END_FUNCTION

FUNCTION _DWORD_TO_REAL:REAL
	VAR_INPUT
		IN :	DWORD;
	END_VAR

	_DWORD_TO_REAL := UDINT_TO_REAL(DWORD_TO_UDINT(IN));

END_FUNCTION

FUNCTION_BLOCK RDM_block
	VAR_INPUT
		LAST :	REAL;
	END_VAR
	VAR_OUTPUT
		RDM :	REAL;
	END_VAR
	VAR
		T_PLC_MS :	T_PLC_MS_block;
		tn :	DWORD;
		tc :	INT;
	END_VAR
	T_PLC_MS();
	tn := UDINT_TO_DWORD(T_PLC_MS.T_PLC_MS);
	tc := Bit_Count(tn);

	tn:=BIT_LOAD_DW(tn,BIT_OF_DWORD(tn,2),31); (* tn.31 := tn.2; *)
	tn:=BIT_LOAD_DW(tn,BIT_OF_DWORD(tn,5),30); (* tn.30 := tn.5; *)
	tn:=BIT_LOAD_DW(tn,BIT_OF_DWORD(tn,4),29); (* tn.29 := tn.4; *)
	tn:=BIT_LOAD_DW(tn,BIT_OF_DWORD(tn,1),28); (* tn.28 := tn.1; *)
	tn:=BIT_LOAD_DW(tn,BIT_OF_DWORD(tn,0),27); (* tn.27 := tn.0; *)
	tn:=BIT_LOAD_DW(tn,BIT_OF_DWORD(tn,7),26); (* tn.26 := tn.7; *)
	tn:=BIT_LOAD_DW(tn,BIT_OF_DWORD(tn,6),25); (* tn.25 := tn.6; *)
	tn:=BIT_LOAD_DW(tn,BIT_OF_DWORD(tn,3),24); (* tn.24 := tn.3; *)

	tn := ROL(tn,Bit_Count(tn)) OR DWORD#16#80000001;
	tn := UDINT_TO_DWORD(DWORD_TO_UDINT(tn) MOD UDINT#71474513 + _INT_TO_UDINT(tc) + UDINT#77);
	RDM := fract(_DWORD_TO_REAL(tn) / 10000000.0 * (2.71828182845904523536028747135266249 - LIMIT_REAL(0.0,last,1.0)));
END_FUNCTION_BLOCK

FUNCTION_BLOCK GEN_RDM_Block

	VAR_INPUT
		PT :	TIME;
		AM :	REAL := REAL#1.0;
		OS :	REAL;
	END_VAR

	VAR_OUTPUT
		Q :	BOOL;
		Out :	REAL;
	END_VAR

	VAR
		tx :	TIME;
		last :	TIME;
		init :	BOOL;
		T_PLC_MS :	T_PLC_MS_Block;
		FB_rdm :	RDM_block;
	END_VAR

	T_PLC_MS();
	tx:= UDINT_TO_TIME(T_PLC_MS.T_PLC_MS) - last;

	IF NOT init THEN
		init := TRUE;
		last := tx;
		tx := t#0s;
	END_IF;

	IF tx >= pt THEN
		last := last + pt;
		tx := tx - pt;

		FB_rdm(last:=0.0);
		out := am * (FB_rdm.RDM - 0.5) + os;
		q := TRUE;
	ELSE
		q := FALSE;
	END_IF;

END_FUNCTION_BLOCK

PROGRAM program0
  VAR
	PT :	TIME;
	AM :	REAL := REAL#1.0;
	OS :	REAL;
	Q :	BOOL;
	Out :	REAL;
	func_block : GEN_RDM_Block;
  END_VAR
	func_block.PT  :=PT;
	func_block.AM  :=AM;
	func_block.OS  :=OS;
	func_block();
	Q := func_block.Q;
	Out := func_block.Out;
END_PROGRAM

CONFIGURATION Config0
	VAR_GLOBAL
		PLC_TICKS_PER_SEC :	INT;
		PLC_SYS_TICK_CNT :	DINT;
	END_VAR
	RESOURCE Res0 ON PLC
		TASK task0(INTERVAL := T#20ms,PRIORITY := 0);
		PROGRAM instance0 WITH task0 : program0;
	END_RESOURCE
END_CONFIGURATION

(* ---- GEN_RDT.ST ---- *)
FUNCTION _REAL_TO_UDINT:UDINT
  VAR_INPUT
    X :	REAL;
  END_VAR

  IF REAL_TO_UDINT(0.5) = UDINT#1 THEN
    _REAL_TO_UDINT := REAL_TO_UDINT(x);
  ELSIF X > 0.0 THEN
    _REAL_TO_UDINT := REAL_TO_UDINT(x+0.5);
  ELSIF X < 0.0 THEN
    _REAL_TO_UDINT := REAL_TO_UDINT(x-0.5);
  ELSE
    _REAL_TO_UDINT := UDINT#0;
  END_IF;
END_FUNCTION

FUNCTION REAL_TO_TIME2:TIME
	VAR_INPUT
		IN :	REAL;
	END_VAR

	REAL_TO_TIME2 := DINT_TO_TIME(UDINT_TO_DINT(_REAL_TO_UDINT(IN)));
END_FUNCTION

FUNCTION TIME_TO_REAL1:REAL

VAR_INPUT
	X :	TIME;
END_VAR

TIME_TO_REAL1 := UDINT_TO_REAL(DINT_TO_UDINT(TIME_TO_DINT(X)));
END_FUNCTION

FUNCTION D_TRUNC : DINT
  VAR_INPUT
    x : REAL;
  END_VAR

  D_TRUNC := REAL_TO_DINT(X);
  IF X > 0.0 THEN
  	IF DINT_TO_REAL(D_TRUNC) > X THEN D_TRUNC := D_TRUNC - DINT#1; END_IF;
  ELSE
  	IF DINT_TO_REAL(D_TRUNC) < X THEN D_TRUNC := D_TRUNC + DINT#1; END_IF;
  END_IF;
END_FUNCTION

FUNCTION BIT_COUNT:INT

	VAR_INPUT
		IN :	DWORD;
	END_VAR

	VAR
		in_temp :	DWORD;
	END_VAR

	in_temp := IN;
	WHILE in_temp > DWORD#0 DO
		IF (in_temp AND DWORD#16#00000001) > DWORD#0 THEN Bit_Count := Bit_Count +1; END_IF;
		in_temp := SHR(in_temp,1);
	END_WHILE;

END_FUNCTION

FUNCTION FRACT:REAL
	VAR_INPUT
		X :	REAL;
	END_VAR

	IF ABS(x) < 2.0E9 THEN
		FRACT := x - DINT_TO_REAL(D_TRUNC(x));
	ELSE
		FRACT := 0.0;
	END_IF;

END_FUNCTION

FUNCTION_BLOCK T_PLC_MS_block
	VAR_OUTPUT
		T_PLC_MS :	UDINT;
	END_VAR

	VAR_EXTERNAL
		PLC_TICKS_PER_SEC :	INT;
		PLC_SYS_TICK_CNT :	DINT;
	END_VAR

	VAR
		debug :	BOOL;(*Debug-Mode ON / OFF*)
		N :	INT;(*Debug-Faktor*)
		Offset :	UDINT;(*Debug-Offset*)
		temp :	DWORD := DWORD#1;(*Debug-Offset*)
		mode :	BOOL;(*modus*)
		faktor :	UDINT;(*Systemtakt-Faktor*)
		init :	BOOL;
		v_plc_ticks_per_sec :	UDINT;
		base :	UDINT := UDINT#1000;
	END_VAR

	IF init = FALSE THEN
		v_plc_ticks_per_sec := INT_TO_UDINT(PLC_TICKS_PER_SEC);
		IF v_plc_ticks_per_sec = UDINT#1024 THEN
			faktor := UDINT#1;
			mode := FALSE;
		ELSIF v_plc_ticks_per_sec > UDINT#0 THEN
			IF v_plc_ticks_per_sec <= base THEN
				faktor := base / v_plc_ticks_per_sec;
				mode := FALSE;
			ELSE
				faktor := v_plc_ticks_per_sec / base;
				mode := TRUE;
			END_IF;
		ELSE
			faktor := UDINT#1;
		END_IF;
		init := TRUE;
	END_IF;

	IF mode THEN
		T_PLC_MS := DINT_TO_UDINT(PLC_SYS_TICK_CNT) / faktor;
	ELSE
		T_PLC_MS := DINT_TO_UDINT(PLC_SYS_TICK_CNT) * faktor;
	END_IF;

	IF debug THEN
		T_PLC_MS := (DWORD_TO_UDINT(SHL(UDINT_TO_DWORD(T_PLC_MS),N) OR SHL(temp,N)) - UDINT#1) + Offset;
	END_IF;

END_FUNCTION_BLOCK

FUNCTION BIT_LOAD_DW:DWORD

	VAR_INPUT
		IN :	DWORD;
		VAL :	BOOL;
		POS :	INT;
	END_VAR

	IF val THEN
		BIT_LOAD_DW := in OR SHL(DWORD#1,pos);
	ELSE
		BIT_LOAD_DW := in AND (NOT SHL(DWORD#1,pos));
	END_IF;

END_FUNCTION

FUNCTION BIT_OF_DWORD : BOOL
  VAR_INPUT
    IN : DWORD;
    N : INT;
  END_VAR

  BIT_OF_DWORD := (SHR(in,N) AND 16#00000001) > 0;
  (* from OSCAT library; www.oscat.de  *)
END_FUNCTION

FUNCTION _INT_TO_UDINT:UDINT
	VAR_INPUT
		IN :	INT;
	END_VAR

	_INT_TO_UDINT := DINT_TO_UDINT(INT_TO_DINT(IN));
END_FUNCTION

FUNCTION _DWORD_TO_REAL:REAL
	VAR_INPUT
		IN :	DWORD;
	END_VAR

	_DWORD_TO_REAL := UDINT_TO_REAL(DWORD_TO_UDINT(IN));

END_FUNCTION

FUNCTION_BLOCK RDM_block
	VAR_INPUT
		LAST :	REAL;
	END_VAR
	VAR_OUTPUT
		RDM :	REAL;
	END_VAR
	VAR
		T_PLC_MS :	T_PLC_MS_block;
		tn :	DWORD;
		tc :	INT;
	END_VAR
	T_PLC_MS();
	tn := UDINT_TO_DWORD(T_PLC_MS.T_PLC_MS);
	tc := Bit_Count(tn);

	tn:=BIT_LOAD_DW(tn,BIT_OF_DWORD(tn,2),31); (* tn.31 := tn.2; *)
	tn:=BIT_LOAD_DW(tn,BIT_OF_DWORD(tn,5),30); (* tn.30 := tn.5; *)
	tn:=BIT_LOAD_DW(tn,BIT_OF_DWORD(tn,4),29); (* tn.29 := tn.4; *)
	tn:=BIT_LOAD_DW(tn,BIT_OF_DWORD(tn,1),28); (* tn.28 := tn.1; *)
	tn:=BIT_LOAD_DW(tn,BIT_OF_DWORD(tn,0),27); (* tn.27 := tn.0; *)
	tn:=BIT_LOAD_DW(tn,BIT_OF_DWORD(tn,7),26); (* tn.26 := tn.7; *)
	tn:=BIT_LOAD_DW(tn,BIT_OF_DWORD(tn,6),25); (* tn.25 := tn.6; *)
	tn:=BIT_LOAD_DW(tn,BIT_OF_DWORD(tn,3),24); (* tn.24 := tn.3; *)

	tn := ROL(tn,Bit_Count(tn)) OR DWORD#16#80000001;
	tn := UDINT_TO_DWORD(DWORD_TO_UDINT(tn) MOD UDINT#71474513 + _INT_TO_UDINT(tc) + UDINT#77);
	RDM := fract(_DWORD_TO_REAL(tn) / 10000000.0 * (2.71828182845904523536028747135266249 - LIMIT_REAL(0.0,last,1.0)));
END_FUNCTION_BLOCK

FUNCTION_BLOCK GEN_RDT_Block

	VAR_INPUT
		ENABLE :	BOOL := TRUE;
		MIN_TIME_MS :	TIME := t#1s;
		MAX_TIME_MS :	TIME := t#1.2s;
		TP_Q :	TIME := t#100ms;
	END_VAR

	VAR_OUTPUT
		XQ :	BOOL;
	END_VAR

	VAR
		tonRDMTimer :	TON;
		tof_xQ :	TOF;
		tRDMTime :	TIME;
		rRDMTime :	REAL;
		rdm_1 :	RDM_Block;
	END_VAR

	tonRDMTimer(IN:=Enable,PT:=tRDMTime);
	tof_xQ(IN := tonRDMTimer.Q,PT:=TP_Q);
	XQ := tof_xq.Q;
	IF tonRDMTimer.Q THEN
		xQ := TRUE ;
		rdm_1(last:=rRDMTime);
		rRDMTime:= rdm_1.RDM;

		tRDMTime := REAL_TO_TIME2(rRDMTime * TIME_TO_REAL1(Max_Time_ms - Min_Time_ms) + TIME_TO_REAL1(Min_Time_ms));
		tonRDMTimer (IN:=FALSE);
	END_IF;

END_FUNCTION_BLOCK

PROGRAM program0
  VAR
	ENABLE :	BOOL := TRUE;
	MIN_TIME_MS :	TIME := t#1s;
	MAX_TIME_MS :	TIME := t#1.2s;
	TP_Q :	TIME := t#100ms;
	XQ :	BOOL;
	func_block : GEN_RDT_Block;
  END_VAR
	func_block.ENABLE  :=ENABLE;
	func_block.MIN_TIME_MS  :=MIN_TIME_MS;
	func_block.MAX_TIME_MS  :=MAX_TIME_MS;
	func_block.TP_Q  :=TP_Q;
	func_block();
	XQ := func_block.XQ;
END_PROGRAM

CONFIGURATION Config0
	VAR_GLOBAL
		PLC_TICKS_PER_SEC :	INT;
		PLC_SYS_TICK_CNT :	DINT;
	END_VAR
	RESOURCE Res0 ON PLC
		TASK task0(INTERVAL := T#20ms,PRIORITY := 0);
		PROGRAM instance0 WITH task0 : program0;
	END_RESOURCE
END_CONFIGURATION

(* ---- GEN_SQ.ST ---- *)
FUNCTION UDINT_TO_TIME2:TIME

	VAR_INPUT
		IN :	UDINT;
	END_VAR

	UDINT_TO_TIME2 := DINT_TO_TIME(UDINT_TO_DINT(IN));

END_FUNCTION

FUNCTION_BLOCK T_PLC_MS_block
	VAR_OUTPUT
		T_PLC_MS :	UDINT;
	END_VAR

	VAR_EXTERNAL
		PLC_TICKS_PER_SEC :	INT;
		PLC_SYS_TICK_CNT :	DINT;
	END_VAR

	VAR
		debug :	BOOL;(*Debug-Mode ON / OFF*)
		N :	INT;(*Debug-Faktor*)
		Offset :	UDINT;(*Debug-Offset*)
		temp :	DWORD := DWORD#1;(*Debug-Offset*)
		mode :	BOOL;(*modus*)
		faktor :	UDINT;(*Systemtakt-Faktor*)
		init :	BOOL;
		v_plc_ticks_per_sec :	UDINT;
		base :	UDINT := UDINT#1000;
	END_VAR

	IF init = FALSE THEN
		v_plc_ticks_per_sec := INT_TO_UDINT(PLC_TICKS_PER_SEC);
		IF v_plc_ticks_per_sec = UDINT#1024 THEN
			faktor := UDINT#1;
			mode := FALSE;
		ELSIF v_plc_ticks_per_sec > UDINT#0 THEN
			IF v_plc_ticks_per_sec <= base THEN
				faktor := base / v_plc_ticks_per_sec;
				mode := FALSE;
			ELSE
				faktor := v_plc_ticks_per_sec / base;
				mode := TRUE;
			END_IF;
		ELSE
			faktor := UDINT#1;
		END_IF;
		init := TRUE;
	END_IF;

	IF mode THEN
		T_PLC_MS := DINT_TO_UDINT(PLC_SYS_TICK_CNT) / faktor;
	ELSE
		T_PLC_MS := DINT_TO_UDINT(PLC_SYS_TICK_CNT) * faktor;
	END_IF;

	IF debug THEN
		T_PLC_MS := (DWORD_TO_UDINT(SHL(UDINT_TO_DWORD(T_PLC_MS),N) OR SHL(temp,N)) - UDINT#1) + Offset;
	END_IF;

END_FUNCTION_BLOCK

FUNCTION_BLOCK GEN_SQ_Block

	VAR_INPUT
		PT :	TIME;
	END_VAR

	VAR_OUTPUT
		Q :	BOOL;
	END_VAR

	VAR
		init :	BOOL;
		tn :	TIME;
		tx :	TIME;
		T_PLC_MS :	T_PLC_MS_Block;
	END_VAR

	T_PLC_MS();
	tx := UDINT_TO_TIME(T_PLC_MS.T_PLC_MS);

	IF NOT init THEN
		init := TRUE;
		tn := tx;
		Q := TRUE;
	ELSIF tx - tn >= DWORD_TO_TIME(SHR(TIME_TO_DWORD(PT),1)) THEN
		Q := NOT Q;
		tn := tn + DWORD_TO_TIME(SHR(TIME_TO_DWORD(pt),1));
	END_IF;

END_FUNCTION_BLOCK

PROGRAM program0
  VAR
	PT :	TIME;
	Q :	BOOL;
	OUT :	REAL;
	func_block : GEN_SQ_Block;
  END_VAR
	func_block.PT  :=PT;
	func_block();
	Q := func_block.Q;
END_PROGRAM

CONFIGURATION Config0
	VAR_GLOBAL
		PLC_TICKS_PER_SEC :	INT;
		PLC_SYS_TICK_CNT :	DINT;
	END_VAR
	RESOURCE Res0 ON PLC
		TASK task0(INTERVAL := T#20ms,PRIORITY := 0);
		PROGRAM instance0 WITH task0 : program0;
	END_RESOURCE
END_CONFIGURATION

(* ---- HEAT_TEMP.ST ---- *)
FUNCTION_BLOCK HEAT_TEMP_Block

	VAR_INPUT
		T_EXT :	REAL;
		T_INT :	REAL;
		OFFSET :	REAL;
		T_REQ :	REAL;
		TY_MAX :	REAL := REAL#70.0;
		TY_MIN :	REAL := REAL#25.0;
		TY_CONFIG :	REAL := REAL#70.0;
		T_INT_CONFIG :	REAL := REAL#20.0;
		T_EXT_CONFIG :	REAL := REAL#-15.0;
		T_DIFF :	REAL := REAL#10.0;
		C :	REAL := REAL#1.33;
		H :	REAL := REAL#3.0;
	END_VAR

	VAR_OUTPUT
		TY :	REAL;
		HEAT :	BOOL;
	END_VAR

	VAR
		tr :	REAL;
		tx :	REAL;
	END_VAR

	tr := T_INT + OFFSET;
	tx := (tr - T_EXT) / (T_INT_CONFIG - T_EXT_CONFIG);

	IF T_EXT + H > tr THEN
		TY := 0.0;
	ELSE
		TY := LIMIT(TY_MIN, tr + T_DIFF * 0.5 * tx + (TY_CONFIG - T_DIFF * 0.5 - tr) * EXPT(tx, 1.0 / C), TY_MAX);
	END_IF;

	TY := MAX(TY, T_REQ);
	HEAT := TY > 0.0;

END_FUNCTION_BLOCK

PROGRAM program0
	VAR
		T_EXT :	REAL;
		T_INT :	REAL;
		OFFSET :	REAL;
		T_REQ :	REAL;
		TY_MAX :	REAL := REAL#70.0;
		TY_MIN :	REAL := REAL#25.0;
		TY_CONFIG :	REAL := REAL#70.0;
		T_INT_CONFIG :	REAL := REAL#20.0;
		T_EXT_CONFIG :	REAL := REAL#-15.0;
		T_DIFF :	REAL := REAL#10.0;
		C :	REAL := REAL#1.33;
		H :	REAL := REAL#3.0;
		TY :	REAL;
		HEAT :	BOOL;

		func_block : HEAT_TEMP_Block;
	END_VAR
	func_block.T_EXT := T_EXT;
	func_block.T_INT := T_INT;
	func_block.OFFSET := OFFSET ;
	func_block.T_REQ    := T_REQ    ;
	func_block.TY_MAX := TY_MAX;
	func_block.TY_MIN := TY_MIN;
	func_block.TY_CONFIG := TY_CONFIG ;
	func_block.T_INT_CONFIG := T_INT_CONFIG ;
	func_block.T_EXT_CONFIG    := T_EXT_CONFIG    ;
	func_block.T_DIFF    := T_DIFF    ;
	func_block.C := C;
	func_block.H := H;

	func_block();
	TY  := func_block.TY;
	HEAT  := func_block.HEAT;
END_PROGRAM

CONFIGURATION Config0
	RESOURCE Res0 ON PLC
		TASK task0(INTERVAL := T#20ms,PRIORITY := 0);
		PROGRAM instance0 WITH task0 : program0;
	END_RESOURCE
END_CONFIGURATION

(* ---- HOLIDAY.ST ---- *)
TYPE oscat_LANGUAGE:
  STRUCT
    DEFAULT 	: INT;
	LMAX    	: INT;
  END_STRUCT;
END_TYPE

TYPE
	oscat_LOCATION_ELEMENTS	: ARRAY [1..5] OF INT;
END_TYPE

TYPE
  oscat_ELEMENT_WEEKDAYS	: ARRAY [1..7] OF STRING;
  oscat_WEEKDAYS			: ARRAY [1..3]  OF oscat_ELEMENT_WEEKDAYS := [0, 0, 0];
END_TYPE

TYPE oscat_LOCATION:
  STRUCT
    DEFAULT 	: INT;
	LMAX    	: INT;
	LANGUAGE	: oscat_LOCATION_ELEMENTS;
  END_STRUCT;
END_TYPE

TYPE oscat_HOLIDAY_DATA :
  STRUCT
	NAME : STRING;
	DAY : SINT;
	MONTH : SINT;
	USE : SINT;
	PAD_BYTE : BYTE;
  END_STRUCT;
END_TYPE

TYPE
  oscat_HOLIDAY_DATA_0_29 	: ARRAY [0..29] OF oscat_HOLIDAY_DATA;
  oscat_HOLIDAY_DATA_0_49 	: ARRAY [0..49] OF oscat_HOLIDAY_DATA;
END_TYPE

FUNCTION_BLOCK SETUP_LANGUAGE_Block

	VAR_IN_OUT
		LANGUAGE :	oscat_LANGUAGE;
	END_VAR

	VAR
		init :	BOOL;
	END_VAR

	IF init THEN RETURN; END_IF;
	init := TRUE;

	LANGUAGE.DEFAULT  := 1; (* 1=english, 2=german 3=french *)
	LANGUAGE.LMAX := 3;
END_FUNCTION_BLOCK

FUNCTION_BLOCK SETUP_LOCATION
	VAR_IN_OUT
		LOCATION :	oscat_LOCATION;
	END_VAR

	VAR
		init :	BOOL;
	END_VAR

	IF init THEN RETURN; END_IF;
	init := TRUE;

	LOCATION.DEFAULT  := 1;
	LOCATION.LMAX := 5;

	LOCATION.LANGUAGE[1] := 2;
	LOCATION.LANGUAGE[2] := 2;
	LOCATION.LANGUAGE[3] := 3;
	LOCATION.LANGUAGE[4] := 2;
	LOCATION.LANGUAGE[5] := 2;
END_FUNCTION_BLOCK

FUNCTION_BLOCK SETUP_WEEKDAYS

	VAR_IN_OUT
		WEEKDAYS :	oscat_WEEKDAYS;
	END_VAR

	VAR
		init :	BOOL;
	END_VAR

	IF init THEN RETURN; END_IF;
	init := TRUE;

	WEEKDAYS[1][01] := 'Monday';
	WEEKDAYS[1][02] := 'Tuesday';
	WEEKDAYS[1][03] := 'Wednesday';
	WEEKDAYS[1][04] := 'Thursday';
	WEEKDAYS[1][05] := 'Friday';
	WEEKDAYS[1][06] := 'Saturday';
	WEEKDAYS[1][07] := 'Sunday';

	WEEKDAYS[2][01] := 'Montag';
	WEEKDAYS[2][02] := 'Dienstag';
	WEEKDAYS[2][03] := 'Mittwoch';
	WEEKDAYS[2][04] := 'Donnerstag';
	WEEKDAYS[2][05] := 'Freitag';
	WEEKDAYS[2][06] := 'Samstag';
	WEEKDAYS[2][07] := 'Sonntag';

	WEEKDAYS[3][01] := 'Lundi';
	WEEKDAYS[3][02] := 'Mardi';
	WEEKDAYS[3][03] := 'Mercredi';
	WEEKDAYS[3][04] := 'Jeudi';
	WEEKDAYS[3][05] := 'Vendredi';
	WEEKDAYS[3][06] := 'Samedi';
	WEEKDAYS[3][07] := 'Dimanche';
END_FUNCTION_BLOCK

FUNCTION YEAR_OF_DATE:INT
	VAR_INPUT
		IDATE :	UDINT;
	END_VAR

	YEAR_OF_DATE := UDINT_TO_INT((idate+UDINT#43200) / UDINT#31557600 + UDINT#1970);
END_FUNCTION

FUNCTION _INT_TO_UDINT:UDINT
	VAR_INPUT
		IN :	INT;
	END_VAR

	_INT_TO_UDINT := DINT_TO_UDINT(INT_TO_DINT(IN));
END_FUNCTION

FUNCTION SET_DATE:UDINT

	VAR_INPUT
		YEAR :	INT;
		MONTH :	INT;
		DAY :	INT;
	END_VAR

	VAR
		count :	INT;
	END_VAR

	IF month > 2 THEN
		count := (month - 1) * 30;
		IF month > 7 THEN
			count := count + DWORD_TO_INT(SHR(DINT_TO_DWORD(INT_TO_DINT(month) - INT_TO_DINT(3)),1));
		ELSE
			count := count + DWORD_TO_INT(SHR(DINT_TO_DWORD(INT_TO_DINT(month) - INT_TO_DINT(4)),1));
		END_IF;
		IF SHL(INT_TO_WORD(year),14) = WORD#0 THEN
			count := count + 1;
		END_IF;
	ELSE
		count := (month - 1) * 31;
	END_IF;
	SET_DATE := (_INT_TO_UDINT(count + day - 1) + DWORD_TO_UDINT(SHR(UDINT_TO_DWORD(_INT_TO_UDINT(year) * UDINT#1461 - UDINT#2878169), 2))) * UDINT#86400;
END_FUNCTION

FUNCTION DAY_OF_WEEK:INT
	VAR_INPUT
		IDATE :	UDINT;
	END_VAR

	DAY_OF_WEEK := UDINT_TO_INT((idate / UDINT#86400 + UDINT#3) MOD UDINT#7) + INT#01;
END_FUNCTION

FUNCTION EASTER:UDINT
	VAR_INPUT
		YEAR :	INT;
	END_VAR

	VAR
		b :	INT;
		c :	INT;
		oday :	INT;
	END_VAR

	b := (204 - 11 * (year MOD 19)) MOD 30;
	IF b > 27 THEN b := b - 1; END_IF;
	c := (year + WORD_TO_INT(SHR(INT_TO_WORD(year),2)) + b - 13) MOD 7;
	oday := 28 + b - c;
	IF oday > 33 THEN
		easter := set_Date(year, 4, oday - 31);
	ELSE
		easter := set_Date(year, 3, oday);
	END_IF;
END_FUNCTION

FUNCTION LEAP_OF_DATE:BOOL

	VAR_INPUT
		IDATE :	UDINT;
	END_VAR

	LEAP_OF_DATE := SHL(UDINT_TO_DWORD((idate + UDINT#43200) / UDINT#31557600), 30) = DWORD#16#80000000;
END_FUNCTION

FUNCTION DAY_OF_YEAR:INT
	VAR_INPUT
		IDATE :	UDINT;
	END_VAR

	DAY_OF_YEAR := UDINT_TO_INT(((idate) / UDINT#86400) MOD UDINT#1461);
	IF DAY_OF_YEAR > 729 THEN
		IF DAY_OF_YEAR > 1095 THEN DAY_OF_YEAR := DAY_OF_YEAR - 1095; ELSE DAY_OF_YEAR := DAY_OF_YEAR - 729; END_IF;
	ELSIF DAY_OF_YEAR > 364 THEN
		DAY_OF_YEAR := DAY_OF_YEAR - 364;
	ELSE
		DAY_OF_YEAR := DAY_OF_YEAR + 1;
	END_IF;
END_FUNCTION

FUNCTION MONTH_OF_DATE:INT

	VAR_INPUT
		IDATE :	UDINT;
	END_VAR

	MONTH_OF_DATE := DAY_OF_YEAR(idate);
	IF MONTH_OF_DATE < 32 THEN
		MONTH_OF_DATE := 1;
	ELSIF LEAP_OF_DATE((IDATE)) THEN
		MONTH_OF_DATE := (MONTH_OF_DATE * 53 + 1668) / 1623;
	ELSE
		MONTH_OF_DATE := (MONTH_OF_DATE * 53 + 1700) / 1620;
	END_IF;
END_FUNCTION

FUNCTION DAY_OF_MONTH:INT
	VAR_INPUT
		IDATE :	UDINT;
	END_VAR

	day_of_month := day_of_year(idate);

	IF leap_of_Date((idate)) THEN
		CASE day_of_month OF
			32..60	:	day_of_month := day_of_month - 31;
			61..91	:	day_of_month := day_of_month - 60;
			92..121 :	day_of_month := day_of_month - 91;
			122..152:	day_of_month := day_of_month - 121;
			153..182:	day_of_month := day_of_month - 152;
			183..213:	day_of_month := day_of_month - 182;
			214..244:	day_of_month := day_of_month - 213;
			245..274:	day_of_month := day_of_month - 244;
			275..305:	day_of_month := day_of_month - 274;
			306..335:	day_of_month := day_of_month - 305;
			336..366:	day_of_month := day_of_month - 335;
		END_CASE;
	ELSE
		CASE day_of_month OF
			32..59	:	day_of_month := day_of_month - 31;
			60..90	:	day_of_month := day_of_month - 59;
			91..120 :	day_of_month := day_of_month - 90;
			121..151:	day_of_month := day_of_month - 120;
			152..181:	day_of_month := day_of_month - 151;
			182..212:	day_of_month := day_of_month - 181;
			213..243:	day_of_month := day_of_month - 212;
			244..273:	day_of_month := day_of_month - 243;
			274..304:	day_of_month := day_of_month - 273;
			305..334:	day_of_month := day_of_month - 304;
			335..365:	day_of_month := day_of_month - 334;
		END_CASE;
	END_IF;
END_FUNCTION

FUNCTION DATE_ADD:UDINT
	VAR_INPUT
		IDATE :	UDINT;
		D :	INT;
		W :	INT;
		M :	INT;
		Y :	INT;
	END_VAR

	VAR
		mo :	INT;
		yr :	INT;
		dm :	INT;
	END_VAR

	DATE_ADD := IDATE + INT_TO_UDINT(D + W * 7) * UDINT#86400;
	yr := Y + YEAR_OF_DATE(DATE_ADD);
	mo := M + MONTH_OF_DATE(DATE_ADD);
	dm := DAY_OF_MONTH(DATE_ADD);
	WHILE mo > 12 DO
		mo := mo - 12;
		yr := yr + 1;
	END_WHILE;
	WHILE mo < 1 DO
		mo := mo + 12;
		yr := yr - 1;
	END_WHILE;
	DATE_ADD := SET_DATE(yr, mo, dm);
END_FUNCTION

FUNCTION_BLOCK HOLIDAY_Block
	VAR_INPUT
		DATE_IN :	UDINT;
		LANGU :	INT;
		FRIDAY :	BOOL;
		SATURDAY :	BOOL;
		SUNDAY :	BOOL;
	END_VAR

	VAR_IN_OUT
		HOLIDAYS :	oscat_HOLIDAY_DATA_0_29;
	END_VAR

	VAR_OUTPUT
		Y :	BOOL;
		NAME :	STRING;
	END_VAR

	VAR
		size :	INT := INT#29;
		last_active :	UDINT;
		ostern :	UDINT;
		i :	INT;
		jahr :	INT;
		x_date :	UDINT;
		lx :	INT;
		wdx :	INT;
		SETUP_LOCATIONS :	SETUP_LOCATION;
		SETUP_WEEKDAYSS :	SETUP_WEEKDAYS;
		SETUP_LANGUAGES :	SETUP_LANGUAGE_Block;
		LOCATION :	oscat_LOCATION;
		WEEKDAYS :	oscat_WEEKDAYS;
		LANGUAGE :	oscat_LANGUAGE;
		wd :	INT;
	END_VAR

	IF last_active = date_in THEN RETURN; END_IF;
	last_active := DATE_IN;

	SETUP_LOCATIONS(LOCATION:=LOCATION);
	LOCATION:=SETUP_LOCATIONS.LOCATION;

	SETUP_WEEKDAYSS(WEEKDAYS:=WEEKDAYS);
	WEEKDAYS:=SETUP_WEEKDAYSS.WEEKDAYS;

	SETUP_LANGUAGES(LANGUAGE:=LANGUAGE);
	LANGUAGE:=SETUP_LANGUAGES.LANGUAGE;

	IF LANGU = 0 THEN
		lx := language.DEFAULT;
	ELSE
		lx := MIN(language.LMAX, LANGU);
	END_IF;

	jahr := YEAR_OF_DATE(date_in);
	ostern := EASTER(jahr);
	wdx := DAY_OF_WEEK(DATE_IN);
	Y := FALSE;

	FOR i := 0 TO size DO
		x_date := SET_DATE(jahr, SINT_TO_INT(HOLIDAYS[i].MONTH) , SINT_TO_INT(HOLIDAYS[i].DAY));
		IF HOLIDAYS[i].USE = SINT#1 AND HOLIDAYS[i].MONTH > SINT#0 THEN
			(* check for fixed date holiday *)
			IF x_date = date_in THEN
				Y := TRUE;
				NAME := HOLIDAYS[i].NAME;
				RETURN;
			END_IF;
		ELSIF HOLIDAYS[i].USE = SINT#1 AND HOLIDAYS[i].MONTH = SINT#0 THEN
			(* check for holiday in reference to easter *)
			IF DATE_ADD(ostern, SINT_TO_INT(HOLIDAYS[i].DAY),0,0,0) = date_in THEN
				Y := TRUE;
				NAME := HOLIDAYS[i].NAME;
				RETURN;
			END_IF;
		ELSIF HOLIDAYS[i].USE < SINT#0 THEN
			(* check for holiday on a weekday before date *)
			IF DAY_OF_WEEK(date_in) = SINT_TO_INT(ABS(HOLIDAYS[i].USE)) AND date_in < x_date AND date_in >= DATE_ADD(x_date,-7,0,0,0) THEN
				Y := TRUE;
				NAME := HOLIDAYS[i].NAME;
				RETURN;
			END_IF;
		END_IF;
	END_FOR;

	IF NOT Y AND (wdx = 5 AND FRIDAY OR wdx = 6 AND SATURDAY OR wdx = 7 AND SUNDAY) THEN
		Y := TRUE;
		wd := LOCATION.LANGUAGE[lx];
		NAME := WEEKDAYS[wd][wdx];
	ELSE
		NAME := '';
	END_IF;
END_FUNCTION_BLOCK

PROGRAM program0
  VAR
	DATE_IN  :	UDINT;
	LANGU    :	INT;
	FRIDAY   :	BOOL;
	SATURDAY :	BOOL;
	SUNDAY   :	BOOL;

	Y :	BOOL;
	NAME :	STRING;

	HOLIDAYS :	oscat_HOLIDAY_DATA_0_29;

	func_block : HOLIDAY_Block;
  END_VAR
	func_block.DATE_IN :=DATE_IN ;
	func_block.LANGU   :=LANGU   ;
	func_block.FRIDAY  :=FRIDAY  ;
	func_block.SATURDAY:=SATURDAY;
	func_block.SUNDAY  :=SUNDAY  ;
	func_block.HOLIDAYS  :=HOLIDAYS ;

	func_block();
	Y := func_block.Y;
	NAME := func_block.NAME;
	HOLIDAYS := func_block.HOLIDAYS;

END_PROGRAM

CONFIGURATION Config0
  RESOURCE Res0 ON PLC
    TASK task0(INTERVAL := T#20ms,PRIORITY := 0);
    PROGRAM instance0 WITH task0 : program0;
  END_RESOURCE
END_CONFIGURATION

(* ---- HYST.ST ---- *)
FUNCTION_BLOCK HYST_Block

	VAR_INPUT
		IN :	REAL;
		_ON :	REAL;
		OFF :	REAL;
	END_VAR

	VAR_OUTPUT
		Q :	BOOL;
		WIN :	BOOL;
	END_VAR

	IF _ON >= OFF THEN
		IF IN < OFF THEN
			Q := FALSE;
			WIN := FALSE;
		ELSIF  IN > _ON THEN
			Q := TRUE;
			WIN := FALSE;
		ELSE
			WIN := TRUE;
		END_IF;
	ELSE
		IF IN > OFF THEN
			Q := FALSE;
			WIN := FALSE;
		ELSIF  IN < _ON THEN
			Q := TRUE;
			WIN := FALSE;
		ELSE
			WIN := TRUE;
		END_IF;
	END_IF;

END_FUNCTION_BLOCK

PROGRAM program0
	VAR
		IN :	REAL;
		_ON :	REAL;
		OFF :	REAL;
		Q :	BOOL;
		WIN :	BOOL;
		func_block : HYST_Block;
	END_VAR
	func_block.IN := IN;
	func_block._ON := _ON;
	func_block.OFF := OFF ;
	func_block();
	Q  := func_block.Q;
	WIN  := func_block.WIN;
END_PROGRAM

CONFIGURATION Config0
	RESOURCE Res0 ON PLC
		TASK task0(INTERVAL := T#20ms,PRIORITY := 0);
		PROGRAM instance0 WITH task0 : program0;
	END_RESOURCE
END_CONFIGURATION

(* ---- HYST_1.ST ---- *)
FUNCTION_BLOCK HYST_1_Block

	VAR_INPUT
		IN :	REAL;
		HIGH :	REAL;
		LOW :	REAL;
	END_VAR

	VAR_OUTPUT
		Q :	BOOL;
		WIN :	BOOL;
	END_VAR

	IF in < low THEN
		Q := FALSE;
		win := FALSE;
	ELSIF in > high THEN
		Q := TRUE;
		win := FALSE;
	ELSE
		win := TRUE;
	END_IF;

END_FUNCTION_BLOCK

PROGRAM program0
	VAR
		IN :	REAL;
		HIGH :	REAL;
		LOW :	REAL;
		Q :	BOOL;
		WIN :	BOOL;
		func_block : HYST_1_Block;
	END_VAR
	func_block.IN := IN;
	func_block.HIGH := HIGH;
	func_block.LOW := LOW;
	func_block();
	Q  := func_block.Q;
	WIN  := func_block.WIN;
END_PROGRAM

CONFIGURATION Config0
	RESOURCE Res0 ON PLC
		TASK task0(INTERVAL := T#20ms,PRIORITY := 0);
		PROGRAM instance0 WITH task0 : program0;
	END_RESOURCE
END_CONFIGURATION

(* ---- HYST_2.ST ---- *)
FUNCTION_BLOCK HYST_2_Block

	VAR_INPUT
		IN :	REAL;
		VAL :	REAL;
		HYS :	REAL;
	END_VAR

	VAR_OUTPUT
		Q :	BOOL;
		WIN :	BOOL;
	END_VAR

	VAR
		tmp :	REAL;
	END_VAR

	tmp := val - hys * 0.5;
	IF in < tmp THEN
		Q := FALSE;
		win := FALSE;
	ELSIF in > tmp + hys THEN
		Q := TRUE;
		win := FALSE;
	ELSE
		win := TRUE;
	END_IF;

END_FUNCTION_BLOCK

PROGRAM program0
	VAR
		IN :	REAL;
		VAL :	REAL;
		HYS :	REAL;
		Q :	BOOL;
		WIN :	BOOL;
		func_block : HYST_2_Block;
	END_VAR
	func_block.IN := IN;
	func_block.VAL := VAL;
	func_block.HYS := HYS;
	func_block();
	Q  := func_block.Q;
	WIN  := func_block.WIN;
END_PROGRAM

CONFIGURATION Config0
	RESOURCE Res0 ON PLC
		TASK task0(INTERVAL := T#20ms,PRIORITY := 0);
		PROGRAM instance0 WITH task0 : program0;
	END_RESOURCE
END_CONFIGURATION

(* ---- HYST_3.ST ---- *)
FUNCTION_BLOCK HYST_3_Block

	VAR_INPUT
		IN :	REAL;
		HYST :	REAL;
		VAL1 :	REAL;
		VAL2 :	REAL;
	END_VAR

	VAR_OUTPUT
		Q1 :	BOOL;
		Q2 :	BOOL;
	END_VAR

	VAR
		X :	REAL;
	END_VAR

	X := hyst * 0.5;
	IF in < val1 - X THEN
		q1 := TRUE;
	ELSIF in > val1 + X THEN
		q1 := FALSE;
	END_IF;
	IF in < val2 - X THEN
		q2 := FALSE;
	ELSIF in > val2 + X THEN
		q2 := TRUE;
	END_IF;

END_FUNCTION_BLOCK

PROGRAM program0
	VAR
		IN :	REAL;
		HYST :	REAL;
		VAL1 :	REAL;
		VAL2 :	REAL;
		Q1 :	BOOL;
		Q2 :	BOOL;
		func_block : HYST_3_Block;
	END_VAR
	func_block.IN := IN;
	func_block.HYST := HYST;
	func_block.VAL1 := VAL1;
	func_block.VAL2 := VAL2;
	func_block();
	Q1  := func_block.Q1;
	Q2  := func_block.Q2;
END_PROGRAM

CONFIGURATION Config0
	RESOURCE Res0 ON PLC
		TASK task0(INTERVAL := T#20ms,PRIORITY := 0);
		PROGRAM instance0 WITH task0 : program0;
	END_RESOURCE
END_CONFIGURATION
